(* CoDeSys 2.3.9.41 project: PLC.pro *)
(* Libraries: ModBus.lib 27.5.09 10:22:38, ComService.lib 21.5.09 15:28:28, SysLibCom.lib 20.2.06 14:31:08, STANDARD.LIB 4.10.05 11:14:46, IECSFC.LIB 13.4.06 15:51:28, SYSLIBTIME.LIB 20.2.06 14:31:16, SYSTASKINFO.LIB 20.2.06 14:31:38, ANALYZATION.LIB 5.10.99 09:05:06, Util.lib 18.5.10 15:14:28, SYSLIBCALLBACK.LIB 20.2.06 14:31:08 *)

(* PLC configuration (modules and I/O channels)
PDI1Q AT %IX0.0 [BitInput] Discrete input 1
PDI2Q AT %IX0.1 [BitInput] Discrete input 2
PDI3Q AT %IX0.2 [BitInput] Discrete input 3
PDI4Q AT %IX0.3 [BitInput] Discrete input 4
Discrete inputs [ID130] node 1, in %IB1 out %QB1 {Filtrationtime_GeneralINP = 10; Visibility = No; PinCount = 12}
  AT %IB1.0 [ByteInput] 8 discrete inputs
  AT %IB1.1 [ByteInput] 4 discrete inputs
Discrete outputs [ID131] node 2, in %IB2 out %QB2 {SafeValueByte = 0; SafeValueByteM = 0; Visibility = No; PinCount = 12}
  AT %QB2.0 [ByteOutput] 8 discrete outputs
  AT %QB2.1 [ByteOutput] 4 discrete outputs
Fast analog inputs [ID125] node 3, in %IB3 out %QB3 {Flt_Comm = 50Hz 2Por}
  AT %IR3.0 [FloatInputP] AI #1 {AIN_TYPE = 4-20 mA; Peak_Filtr = 200; Flt_Ch = Off; TauRC = 10; MinFV = 0; MaxFV = 20000.0}
  AT %IR3.1 [FloatInputP] AI #2 {AIN_TYPE = 4-20 mA; Peak_Filtr = 200; Flt_Ch = Off; TauRC = 10; MinFV = 0; MaxFV = 20000.0}
  AT %IR3.2 [FloatInputP] AI #3 {AIN_TYPE = 4-20 mA; Peak_Filtr = 200; Flt_Ch = Off; TauRC = 10; MinFV = 0; MaxFV = 20000.0}
  AT %IR3.3 [FloatInputP] AI #4 {AIN_TYPE = 4-20 mA; Peak_Filtr = 200; Flt_Ch = Off; TauRC = 10; MinFV = 0; MaxFV = 20000.0}
  AT %IR3.4 [FloatInputP] AI #5 {AIN_TYPE = 4-20 mA; Peak_Filtr = 200; Flt_Ch = Off; TauRC = 10; MinFV = 0; MaxFV = 20000.0}
  AT %IR3.5 [FloatInputP] AI #6 {AIN_TYPE = 4-20 mA; Peak_Filtr = 200; Flt_Ch = Off; TauRC = 10; MinFV = 0; MaxFV = 20000.0}
  AT %IR3.6 [FloatInputP] AI #7 {AIN_TYPE = 4-20 mA; Peak_Filtr = 200; Flt_Ch = Off; TauRC = 10; MinFV = 0; MaxFV = 20000.0}
  AT %IR3.7 [FloatInputP] AI #8 {AIN_TYPE = 4-20 mA; Peak_Filtr = 200; Flt_Ch = Off; TauRC = 10; MinFV = 0; MaxFV = 20000.0}
  AT %IW3.8 [WordInput] AI read time (10ms)
Analog outputs [ID126] node 4, in %IB4 out %QB4
  PAO01 AT %QR4.0 [FloatOutputP] AO #1 {AOUT_TYPE = 4-20 mA; SafeValueREAL = 0.0}
  AT %QR4.1 [FloatOutputP] AO #2 {AOUT_TYPE = 4-20 mA; SafeValueREAL = 0.0}
  AT %QR4.2 [FloatOutputP] AO #3 {AOUT_TYPE = 4-20 mA; SafeValueREAL = 0.0}
  AT %QR4.3 [FloatOutputP] AO #4 {AOUT_TYPE = 4-20 mA; SafeValueREAL = 0.0}
Special input [ID103] node 5, in %IB5 out %QB5 {Filtrationtime = 1000; PinCount = 1; WatchDogPeriod = 400; PollPeriod = 3000; Visibility = No}
  AT %IX5.0 [BitInput] Special input
Special output [ID104] node 6, in %IB6 out %QB6 {Visibility = No; PinCount = 1}
  AT %QX6.0 [BitOutput] Special output
Modbus [MODBUS_ID302] node 0, in %IB7.0 out %QB7.0
  TCP [TCP_ID221] node 0, in %IB7.0.0 out %QB7.0.0 {RemotePort = 502; Visibility = No}
  TCP [TCP_ID221] node 1, in %IB7.0.1 out %QB7.0.1 {RemotePort = 502; Visibility = No}
  TCP [TCP_ID221] node 2, in %IB7.0.2 out %QB7.0.2 {RemotePort = 504; Visibility = No}
  TCP [TCP_ID221] node 3, in %IB7.0.3 out %QB7.0.3 {RemotePort = 502; Visibility = No}
  TCP [TCP_ID221] node 4, in %IB7.0.4 out %QB7.0.4 {RemotePort = 502; Visibility = No}
  RS-232 [COM2_USART] node 5, in %IB7.0.5 out %QB7.0.5 {CommunicationSpeed = 11520; Parity = NO PARITY CHECK; BitLength = 8 bits; StopLength = One stop bit; InterfaceType = RS232; FrameOriented = RTU; Timeout = 0; Visibility = No}
  Debug RS-232 [DEBUG_USART] node 6, in %IB7.0.6 out %QB7.0.6 {CommunicationSpeed = 11520; Parity = NO PARITY CHECK; BitLength = 8 bits; StopLength = One stop bit; InterfaceType = RS232; FrameOriented = RTU; Timeout = 0; Visibility = No}
  TCP [TCP_ID221] node 7, in %IB7.0.7 out %QB7.0.7 {RemotePort = 502; Visibility = No}
  TCP [TCP_ID221] node 8, in %IB7.0.8 out %QB7.0.8 {RemotePort = 502; Visibility = No}
AT %QB7.1.0 [ByteOutput]
8 bits [8Bit] node 2, in %IB7.2 out %QB7.2
  AT %QB7.2.0 [ByteOutput]
8 bits [8Bit] node 3, in %IB7.3 out %QB7.3
  AT %QB7.3.0 [ByteOutput]
8 bits [8Bit] node 4, in %IB7.4 out %QB7.4
  AT %QB7.4.0 [ByteOutput]
  AT %QB7.5.0 [ByteOutput]
8 bits [8Bit] node 6, in %IB7.6 out %QB7.6
  AT %QB7.6.0 [ByteOutput]
  Bit 7 AT %QB7.7.0 [ByteOutput] Module.8Bit3Module.MODBUS_ID4008 bitsIB%QB%MB%M
8 bits [8Bit] node 8, in %IB7.8 out %QB7.8
  AT %QB7.8.0 [ByteOutput]
  AT %QB7.9.0 [ByteOutput]
  AT %QB7.10.0 [ByteOutput]
  AT %QB7.11.0 [ByteOutput]
  AT %QB7.12.0 [ByteOutput]
  AT %QB7.13.0 [ByteOutput]
  AT %QB7.14.0 [ByteOutput]
  AT %QB7.15.0 [ByteOutput]
  AT %QB7.16.0 [ByteOutput]
  AT %QB7.17.0 [ByteOutput]
  AT %QB7.18.0 [ByteOutput]
  AT %QB7.19.0 [ByteOutput]
  AT %QB7.20.0 [ByteOutput]
8 bits [8Bit] node 21, in %IB7.21 out %QB7.21
  AT %QB7.21.0 [ByteOutput]
8 bits [8Bit] node 22, in %IB7.22 out %QB7.22
  AT %QB7.22.0 [ByteOutput]
2 byte [Register] node 23, in %IB7.23 out %QB7.23
  L16001_CUR AT %QW7.23.0 [WordOutput]
2 byte [Register] node 24, in %IB7.24 out %QB7.24
  L16106_CUR AT %QW7.24.0 [WordOutput]
2 byte [Register] node 25, in %IB7.25 out %QB7.25
  X16106M1_CUR AT %QW7.25.0 [WordOutput]
2 byte [Register] node 26, in %IB7.26 out %QB7.26
  C16105_CUR AT %QW7.26.0 [WordOutput]
2 byte [Register] node 27, in %IB7.27 out %QB7.27
  M16105_PER AT %QW7.27.0 [WordOutput]
2 byte [Register] node 28, in %IB7.28 out %QB7.28
  C16103_CUR AT %QW7.28.0 [WordOutput]
2 byte [Register] node 29, in %IB7.29 out %QB7.29
  M16103_PER AT %QW7.29.0 [WordOutput]
2 byte [Register] node 30, in %IB7.30 out %QB7.30
  M16106_PV AT %QW7.30.0 [WordOutput]
2 byte [Register] node 31, in %IB7.31 out %QB7.31
  L16201_CUR AT %QW7.31.0 [WordOutput]
2 byte [Register] node 32, in %IB7.32 out %QB7.32
  X16105A_CUR AT %QW7.32.0 [WordOutput]
2 byte [Register] node 33, in %IB7.33 out %QB7.33
  X16105B_CUR AT %QW7.33.0 [WordOutput]
2 byte [Register] node 34, in %IB7.34 out %QB7.34
  C16104_CUR AT %QW7.34.0 [WordOutput]
2 byte [Register] node 35, in %IB7.35 out %QB7.35
  M16104_PER AT %QW7.35.0 [WordOutput]
2 byte [Register] node 36, in %IB7.36 out %QB7.36
  L16101_CUR AT %QW7.36.0 [WordOutput]
2 byte [Register] node 37, in %IB7.37 out %QB7.37
  TRM_1_1 AT %QW7.37.0 [WordOutput]
2 byte [Register] node 38, in %IB7.38 out %QB7.38
  TRM_1_2 AT %QW7.38.0 [WordOutput]
2 byte [Register] node 39, in %IB7.39 out %QB7.39
  TRM_1_3 AT %QW7.39.0 [WordOutput]
  TRM_1_4 AT %QW7.40.0 [WordOutput]
2 byte [Register] node 41, in %IB7.41 out %QB7.41
  TRM_1_5 AT %QW7.41.0 [WordOutput]
2 byte [Register] node 42, in %IB7.42 out %QB7.42
  TRM_1_6 AT %QW7.42.0 [WordOutput]
2 byte [Register] node 43, in %IB7.43 out %QB7.43
  TRM_1_7 AT %QW7.43.0 [WordOutput]
2 byte [Register] node 44, in %IB7.44 out %QB7.44
  TRM_1_8 AT %QW7.44.0 [WordOutput]
2 byte [Register] node 45, in %IB7.45 out %QB7.45
  TRM_2_1 AT %QW7.45.0 [WordOutput]
2 byte [Register] node 46, in %IB7.46 out %QB7.46
  TRM_2_2 AT %QW7.46.0 [WordOutput]
2 byte [Register] node 47, in %IB7.47 out %QB7.47
  TRM_2_3 AT %QW7.47.0 [WordOutput]
2 byte [Register] node 48, in %IB7.48 out %QB7.48
  TRM_2_4 AT %QW7.48.0 [WordOutput]
2 byte [Register] node 49, in %IB7.49 out %QB7.49
  TRM_2_5 AT %QW7.49.0 [WordOutput]
2 byte [Register] node 50, in %IB7.50 out %QB7.50
  TRM_2_6 AT %QW7.50.0 [WordOutput]
2 byte [Register] node 51, in %IB7.51 out %QB7.51
  TRM_2_7 AT %QW7.51.0 [WordOutput]
2 byte [Register] node 52, in %IB7.52 out %QB7.52
  TRM_2_8 AT %QW7.52.0 [WordOutput]
2 byte [Register] node 53, in %IB7.53 out %QB7.53
  K16001_P AT %QW7.53.0 [WordOutput]
2 byte [Register] node 54, in %IB7.54 out %QB7.54
  M_3_6 AT %QW7.54.0 [WordOutput]
2 byte [Register] node 55, in %IB7.55 out %QB7.55
  M_3_7 AT %QW7.55.0 [WordOutput]
2 byte [Register] node 56, in %IB7.56 out %QB7.56
  M16106_CUR AT %QW7.56.0 [WordOutput]
  M16106_SP AT %QW7.57.0 [WordOutput]
  AT %QW7.58.0 [WordOutput]
2 byte [Register] node 59, in %IB7.59 out %QB7.59
  AT %QW7.59.0 [WordOutput]
2 byte [Register] node 60, in %IB7.60 out %QB7.60
  AT %QW7.60.0 [WordOutput]
2 byte [Register] node 61, in %IB7.61 out %QB7.61
  AT %QW7.61.0 [WordOutput]
2 byte [Register] node 62, in %IB7.62 out %QB7.62
  AT %QW7.62.0 [WordOutput]
2 byte [Register] node 63, in %IB7.63 out %QB7.63
  AT %QW7.63.0 [WordOutput]
2 byte [Register] node 64, in %IB7.64 out %QB7.64
  AT %QW7.64.0 [WordOutput]
2 byte [Register] node 65, in %IB7.65 out %QB7.65
  AT %QW7.65.0 [WordOutput]
  FLOW_SP_1 AT %QW7.66.0 [WordOutput]
  FLOW_SP_2 AT %QW7.67.0 [WordOutput]
  FLOW_SP_3 AT %QW7.68.0 [WordOutput]
  FLOW_SP_4 AT %QW7.69.0 [WordOutput]
  SPEED_1 AT %QW7.70.0 [WordOutput]
  SPEED_2 AT %QW7.71.0 [WordOutput]
  SPEED_3 AT %QW7.72.0 [WordOutput]
  SPEED_4 AT %QW7.73.0 [WordOutput]
  PERSENT1 AT %QW7.74.0 [WordOutput]
  PERSENT2 AT %QW7.75.0 [WordOutput]
  PERSENT3 AT %QW7.76.0 [WordOutput]
  PERSENT4 AT %QW7.77.0 [WordOutput]
  FLOW_TOT AT %QW7.78.0 [WordOutput]
  PER_TOT AT %QW7.79.0 [WordOutput]
  FLOW_SP_TOT AT %QW7.80.0 [WordOutput]
8 bits [8Bit] node 81, in %IB7.81 out %QB7.81
  AT %QB7.81.0 [ByteOutput]
8 bits [8Bit] node 82, in %IB7.82 out %QB7.82
  AT %QB7.82.0 [ByteOutput]
  AT %QB7.83.0 [ByteOutput]
  AT %QB7.84.0 [ByteOutput]
FLOW_1 AT %QW7.85.0 [WordOutput]
FLOW_2 AT %QW7.86.0 [WordOutput]
FLOW_3 AT %QW7.87.0 [WordOutput]
FLOW_4 AT %QW7.88.0 [WordOutput]
counter_1 AT %QD7.89.0 [FloatOutput]
counter_2 AT %QD7.90.0 [FloatOutput]
counter_3 AT %QD7.91.0 [FloatOutput]
counter_4 AT %QD7.92.0 [FloatOutput]
count_hour1 AT %QW7.93.0 [WordOutput]
count_hour2 AT %QW7.94.0 [WordOutput]
count_hour3 AT %QW7.95.0 [WordOutput]
count_hour4 AT %QW7.96.0 [WordOutput]
count_TOTAL AT %QW7.97.0 [WordOutput]
ModBus (Master) [MODBUS_MASTER_ID450] node 8, in %IB8 out %QB8 {Visibility = No}
  AT %QD8.0 [DWordOutput] Last address
  AT %QW8.1 [WordOutput] Last error
  RS-485-1 [COM1_USART] node 0, in %IB8.0 out %QB8.0 {CommunicationSpeed = 9600; Parity = NO PARITY CHECK; BitLength = 8 bits; StopLength = One stop bit; InterfaceType = RS485; FrameOriented = RTU; Timeout = 0; Visibility = No}
AT %QB8.1.0 [ComChannel] Command (0xff - Start)
count1 AT %ID8.1.0.0 [DWordInput]
flow1 AT %ID8.1.1.0 [DWordInput]
flow_sp1 AT %QD8.1.2.0 [DWordOutput]
speed1 AT %ID8.1.3.0 [DWordInput]
start1 AT %QW8.1.4.0 [WordOutput]
STATUS1 AT %IW8.1.5.0 [WordInput]
AT %QB8.2.0 [ComChannel] Command (0xff - Start)
count2 AT %ID8.2.0.0 [DWordInput]
flow2 AT %ID8.2.1.0 [DWordInput]
flow_sp2 AT %QD8.2.2.0 [DWordOutput]
speed2 AT %ID8.2.3.0 [DWordInput]
start2 AT %QW8.2.4.0 [WordOutput]
STATUS2 AT %IW8.2.5.0 [WordInput]
AT %QB8.3.0 [ComChannel] Command (0xff - Start)
count3 AT %ID8.3.0.0 [DWordInput]
flow3 AT %ID8.3.1.0 [DWordInput]
flow_sp3 AT %QD8.3.2.0 [DWordOutput]
speed3 AT %ID8.3.3.0 [DWordInput]
start3 AT %QW8.3.4.0 [WordOutput]
STATUS3 AT %IW8.3.5.0 [WordInput]
AT %QB8.4.0 [ComChannel] Command (0xff - Start)
count4 AT %ID8.4.0.0 [DWordInput]
flow4 AT %ID8.4.1.0 [DWordInput]
flow_sp4 AT %QD8.4.2.0 [DWordOutput]
speed4 AT %ID8.4.3.0 [DWordInput]
start4 AT %QW8.4.4.0 [WordOutput]
STATUS4 AT %IW8.4.5.0 [WordInput]
Universal Modbus device [ID2000] node 5, in %IB8.5 out %QB8.5 {ModuleIP = 10:0:0:223; ServiceTimeout = 150; TCPport = 502; NetMode = Serial; ModuleSlaveAddress = 8; RequestType = Both; PeriodOfService = 10; Visibility = No; RepeatCounter = 0; ByteSequence = Trace_mode}
  AT %QB8.5.0 [ComChannel] Command (0xff - Start)
MDI_1_0 AT %IW8.5.0.0 [WordInput]
MDI_1_1 AT %IW8.5.1.0 [WordInput]
Universal Modbus device [ID2000] node 6, in %IB8.6 out %QB8.6 {ModuleIP = 10:0:0:223; ServiceTimeout = 150; TCPport = 502; NetMode = Serial; ModuleSlaveAddress = 16; RequestType = Both; PeriodOfService = 10; Visibility = No; RepeatCounter = 0; ByteSequence = Trace_mode}
  AT %QB8.6.0 [ComChannel] Command (0xff - Start)
MDI_2_0 AT %IW8.6.0.0 [WordInput]
MDI_2_1 AT %IW8.6.1.0 [WordInput]
Universal Modbus device [ID2000] node 7, in %IB8.7 out %QB8.7 {ModuleIP = 10:0:0:223; ServiceTimeout = 150; TCPport = 502; NetMode = Serial; ModuleSlaveAddress = 24; RequestType = Both; PeriodOfService = 10; Visibility = No; RepeatCounter = 0; ByteSequence = Trace_mode}
  AT %QB8.7.0 [ComChannel] Command (0xff - Start)
MDI_3_0 AT %IW8.7.0.0 [WordInput]
MDI_3_1 AT %IW8.7.1.0 [WordInput]
Universal Modbus device [ID2000] node 8, in %IB8.8 out %QB8.8 {ModuleIP = 10:0:0:223; ServiceTimeout = 150; TCPport = 502; NetMode = Serial; ModuleSlaveAddress = 32; RequestType = Both; PeriodOfService = 10; Visibility = No; RepeatCounter = 0; ByteSequence = Trace_mode}
  AT %QB8.8.0 [ComChannel] Command (0xff - Start)
MDI_4_0 AT %IW8.8.0.0 [WordInput]
MDI_4_1 AT %IW8.8.1.0 [WordInput]
Universal Modbus device [ID2000] node 9, in %IB8.9 out %QB8.9 {ModuleIP = 10:0:0:223; ServiceTimeout = 150; TCPport = 502; NetMode = Serial; ModuleSlaveAddress = 40; RequestType = Both; PeriodOfService = 10; Visibility = No; RepeatCounter = 0; ByteSequence = Trace_mode}
  AT %QB8.9.0 [ComChannel] Command (0xff - Start)
MDO1_0 AT %QW8.9.0.0 [WordOutput]
MDO1_1 AT %QW8.9.1.0 [WordOutput]
MDO1_2 AT %QW8.9.2.0 [WordOutput]
MDO1_3 AT %QW8.9.3.0 [WordOutput]
MDO1_4 AT %QW8.9.4.0 [WordOutput]
MDO1_5 AT %QW8.9.5.0 [WordOutput]
MDO1_6 AT %QW8.9.6.0 [WordOutput]
MDO1_7 AT %QW8.9.7.0 [WordOutput]
MDO1_8 AT %QW8.9.8.0 [WordOutput]
MDO1_9 AT %QW8.9.9.0 [WordOutput]
MDO1_10 AT %QW8.9.10.0 [WordOutput]
MDO1_11 AT %QW8.9.11.0 [WordOutput]
MDO1_12 AT %QW8.9.12.0 [WordOutput]
MDO1_13 AT %QW8.9.13.0 [WordOutput]
MDO1_14 AT %QW8.9.14.0 [WordOutput]
MDO1_15 AT %QW8.9.15.0 [WordOutput]
Universal Modbus device [ID2000] node 10, in %IB8.10 out %QB8.10 {ModuleIP = 10:0:0:223; ServiceTimeout = 150; TCPport = 502; NetMode = Serial; ModuleSlaveAddress = 48; RequestType = Both; PeriodOfService = 10; Visibility = No; RepeatCounter = 0; ByteSequence = Trace_mode}
  AT %QB8.10.0 [ComChannel] Command (0xff - Start)
MDO2_0 AT %QW8.10.0.0 [WordOutput]
MDO2_1 AT %QW8.10.1.0 [WordOutput]
MDO2_2 AT %QW8.10.2.0 [WordOutput]
MDO2_3 AT %QW8.10.3.0 [WordOutput]
MDO2_4 AT %QW8.10.4.0 [WordOutput]
MDO2_5 AT %QW8.10.5.0 [WordOutput]
MDO2_6 AT %QW8.10.6.0 [WordOutput]
MDO2_7 AT %QW8.10.7.0 [WordOutput]
MDO2_8 AT %QW8.10.8.0 [WordOutput]
MDO2_9 AT %QW8.10.9.0 [WordOutput]
MDO2_10 AT %QW8.10.10.0 [WordOutput]
MDO2_11 AT %QW8.10.11.0 [WordOutput]
MDO2_12 AT %QW8.10.12.0 [WordOutput]
MDO2_13 AT %QW8.10.13.0 [WordOutput]
MDO2_14 AT %QW8.10.14.0 [WordOutput]
MDO2_15 AT %QW8.10.15.0 [WordOutput]
Universal Modbus device [ID2000] node 11, in %IB8.11 out %QB8.11 {ModuleIP = 10:0:0:223; ServiceTimeout = 150; TCPport = 502; NetMode = Serial; ModuleSlaveAddress = 56; RequestType = Both; PeriodOfService = 10; Visibility = No; RepeatCounter = 0; ByteSequence = Trace_mode}
  AT %QB8.11.0 [ComChannel] Command (0xff - Start)
M1_1 AT %IW8.11.0.0 [WordInput]
M1_2 AT %IW8.11.1.0 [WordInput]
M1_3 AT %IW8.11.2.0 [WordInput]
M1_4 AT %IW8.11.3.0 [WordInput]
M1_5 AT %IW8.11.4.0 [WordInput]
M1_6 AT %IW8.11.5.0 [WordInput]
M1_7 AT %IW8.11.6.0 [WordInput]
M1_8 AT %IW8.11.7.0 [WordInput]
Universal Modbus device [ID2000] node 12, in %IB8.12 out %QB8.12 {ModuleIP = 10:0:0:223; ServiceTimeout = 150; TCPport = 502; NetMode = Serial; ModuleSlaveAddress = 64; RequestType = Both; PeriodOfService = 10; Visibility = No; RepeatCounter = 0; ByteSequence = Trace_mode}
  AT %QB8.12.0 [ComChannel] Command (0xff - Start)
M2_1 AT %IW8.12.0.0 [WordInput]
M2_2 AT %IW8.12.1.0 [WordInput]
M2_3 AT %IW8.12.2.0 [WordInput]
M2_4 AT %IW8.12.3.0 [WordInput]
M2_5 AT %IW8.12.4.0 [WordInput]
M2_6 AT %IW8.12.5.0 [WordInput]
M2_7 AT %IW8.12.6.0 [WordInput]
M2_8 AT %IW8.12.7.0 [WordInput]
Universal Modbus device [ID2000] node 13, in %IB8.13 out %QB8.13 {ModuleIP = 10:0:0:223; ServiceTimeout = 150; TCPport = 502; NetMode = Serial; ModuleSlaveAddress = 72; RequestType = Both; PeriodOfService = 10; Visibility = No; RepeatCounter = 0; ByteSequence = Trace_mode}
  AT %QB8.13.0 [ComChannel] Command (0xff - Start)
M3_1 AT %IW8.13.0.0 [WordInput]
M3_2 AT %IW8.13.1.0 [WordInput]
M3_3 AT %IW8.13.2.0 [WordInput]
M3_4 AT %IW8.13.3.0 [WordInput]
M3_5 AT %IW8.13.4.0 [WordInput]
M3_6 AT %IW8.13.5.0 [WordInput]
M3_7 AT %IW8.13.6.0 [WordInput]
M3_8 AT %IW8.13.7.0 [WordInput]
Universal Modbus device [ID2000] node 14, in %IB8.14 out %QB8.14 {ModuleIP = 10:0:0:223; ServiceTimeout = 150; TCPport = 502; NetMode = Serial; ModuleSlaveAddress = 80; RequestType = Both; PeriodOfService = 10; Visibility = No; RepeatCounter = 0; ByteSequence = Trace_mode}
  AT %QB8.14.0 [ComChannel] Command (0xff - Start)
TRM_1_1_RS AT %ID8.14.0.0 [FloatInput]
TRM_1_2_RS AT %ID8.14.1.0 [FloatInput]
TRM_1_3_RS AT %ID8.14.2.0 [FloatInput]
TRM_1_4_RS AT %ID8.14.3.0 [FloatInput]
TRM_1_5_RS AT %ID8.14.4.0 [FloatInput]
TRM_1_6_RS AT %ID8.14.5.0 [FloatInput]
TRM_1_7_RS AT %ID8.14.6.0 [FloatInput]
TRM_1_8_RS AT %ID8.14.7.0 [FloatInput]
Universal Modbus device [ID2000] node 15, in %IB8.15 out %QB8.15 {ModuleIP = 10:0:0:223; ServiceTimeout = 150; TCPport = 502; NetMode = Serial; ModuleSlaveAddress = 88; RequestType = Both; PeriodOfService = 10; Visibility = No; RepeatCounter = 0; ByteSequence = Trace_mode}
  AT %QB8.15.0 [ComChannel] Command (0xff - Start)
TRM_2_1_RS AT %ID8.15.0.0 [FloatInput]
TRM_2_2_RS AT %ID8.15.1.0 [FloatInput]
TRM_2_3_RS AT %ID8.15.2.0 [FloatInput]
TRM_2_4_RS AT %ID8.15.3.0 [FloatInput]
TRM_2_5_RS AT %ID8.15.4.0 [FloatInput]
TRM_2_6_RS AT %ID8.15.5.0 [FloatInput]
TRM_2_7_RS AT %ID8.15.6.0 [FloatInput]
TRM_2_8_RS AT %ID8.15.7.0 [FloatInput]
Button [ID003] node 9, in %IB9 out %QB9
  AT %IX9.0 [BitInput] Button Start/Stop
*)

(* Global variable list: Global_Variables *)
VAR_GLOBAL
	L16003_SRT_G : BOOL;
	X16011_SRT_G : BOOL;
	L16106_SRT_G : BOOL;
	L16004_SRT_G : BOOL;
	X16011_A_SRT_G : BOOL;
	X16106M1_SRT_G : BOOL;
	X16106M1_STP_G : BOOL;
	X16106MA_SRT_G : BOOL;
	X16106MB_SRT_G : BOOL;
	X16106M2_SRT_G : BOOL;
	O161061_SRT_G : BOOL;
	O161062_SRT_G : BOOL;
	O161063_SRT_G : BOOL;
	O161064_SRT_G : BOOL;
	C16101_SRT_G : BOOL;
	C16105_SRT_G : BOOL;
	(*********************************)
	M16105_OPN_G : BOOL;
	M16105_CLS_G : BOOL;
	C16103_SRT_G : BOOL;
	M16103_OPN_G : BOOL;
	M16103_CLS_G : BOOL;
	C16106_SRT_G : BOOL;
	L16107_SRT_G : BOOL;
	M16106_SRT_G : BOOL;
	O16106_SRT_G : BOOL;
	B16401_SRT_G : BOOL;
	B16402_SRT_G : BOOL;
	X16106M1_G : BOOL;
	B16404_SRT_G : BOOL;
	L16005_SRT_G : BOOL;

	L16201_SRT_G : BOOL;
	C16201_SRT_G : BOOL;
	(*****************************)
	C16104_SRT_G : BOOL;
	L16101_SRT_G : BOOL;
	X16106M1_FAZA_G : BOOL;

END_VAR
VAR_GLOBAL RETAIN PERSISTENT

	eski_counter_1: REAL;
	eski_counter_2: REAL;
	eski_counter_3: REAL;
	eski_counter_4: REAL;


END_VAR

(* POU PLC_PRG, ST *)
PROGRAM PLC_PRG
VAR
END_VAR
TRANSLATE();
ALARM_RPM();
(*BLOCK();*)
vaqt();
END_PROGRAM

(* POU TRANSLATE, ST *)
PROGRAM TRANSLATE
VAR
	B164: BOOL;
	MA : ARRAY [1..30] OF MY_LINTRAFO;
	RTRIG: R_TRIG;
	FTRIG: F_TRIG;

	FLOW_ZAD: BOOL;
	FLOW_ZAD_1: BOOL;
	FLOW_ZAD_2: BOOL;
	FLOW_ZAD_3: BOOL;
	FLOW_ZAD_4: BOOL;
	f: BOOL;

	PAO01_TMP: WORD;
END_VAR
OUTPUTS();
MDI1_0();
MDI1_1();
MDI2_0();
MDI2_1();
MDI3_0();
MDI3_1();
MDI4_0();
MDI4_1();


DOZ();
BLOCK();
 M16106_SP := LIMIT(10, M16106_SP, 50);
MA[30](IN := M16106_SP,  IN_MIN := 10, IN_MAX :=50 , OUT_MIN := 4.0,  OUT_MAX := 20.0, OUT => PAO01_TMP);
PAO01 := PAO01_TMP / 100.0;
MA[1](IN := M1_1, IN_MIN := 400.0, IN_MAX := 2000.0, OUT_MIN := 0.0,  OUT_MAX := 200.0, OUT => L16001_CUR);
MA[2](IN := M1_2,  OUT_MIN := 0.0,  OUT_MAX := 200.0, OUT => L16106_CUR);
MA[3](IN := M1_7, IN_MIN := 400.0, IN_MAX := 2000.0, OUT_MIN := 0.0,  OUT_MAX := 290.0, OUT => X16106M1_CUR);
MA[4](IN := M1_3, OUT_MIN := 0.0,  OUT_MAX := 200.0, OUT => C16105_CUR);
MA[5](IN := M1_4, IN_MIN := 800, IN_MAX := 2000,  OUT_MIN := 0.0,  OUT_MAX := 100.0, OUT => M16105_PER);
MA[6](IN := M2_7, OUT_MIN :=0.0,  OUT_MAX := 100.0, OUT => C16103_CUR);
MA[7](IN := M2_8, OUT_MIN := 0.0,  OUT_MAX := 100.0, OUT => M16103_PER);
MA[8](IN := M1_6,  IN_MIN := 400.0, IN_MAX := 2000.0, OUT_MIN := 0.0,  OUT_MAX := 50.0, OUT => M16106_CUR);
MA[9](IN := M2_1, OUT_MIN := 0.0,  OUT_MAX := 200.0, OUT => L16201_CUR);
MA[10](IN := M2_4, OUT_MIN := 0.0,  OUT_MAX := 200.0, OUT =>C16104_CUR);
MA[11](IN := M2_5,  IN_MIN := 0.0, IN_MAX := 100.0, OUT_MIN := 0.0,  OUT_MAX := 100.0, OUT => M16104_PER);
MA[12](IN := M2_6, OUT_MIN := 0.0,  OUT_MAX := 200.0, OUT => L16101_CUR);
MA[17](IN := M1_8, IN_MIN := 400.0, IN_MAX := 2000.0, OUT_MIN := 0.0,  OUT_MAX := 496.0, OUT => M16106_PV);
TRM_1_1 := REAL_TO_WORD( TRM_1_1_RS * 100);
TRM_1_2 := REAL_TO_WORD(TRM_1_2_RS * 100);
TRM_1_3 := REAL_TO_WORD(TRM_1_3_RS * 100);
TRM_1_4 := REAL_TO_WORD(TRM_1_4_RS * 100);
TRM_1_5 := REAL_TO_WORD(TRM_1_5_RS * 100);
TRM_1_6 := REAL_TO_WORD(TRM_1_6_RS * 100);
TRM_1_7 := REAL_TO_WORD(TRM_1_7_RS * 100);
TRM_1_8 := REAL_TO_WORD(TRM_1_8_RS * 100);

TRM_2_1 := REAL_TO_WORD(TRM_2_1_RS * 100);
TRM_2_2 := REAL_TO_WORD(TRM_2_2_RS * 100);
TRM_2_3 := REAL_TO_WORD(TRM_2_3_RS * 100);
TRM_2_4 := REAL_TO_WORD(TRM_2_4_RS * 100);
TRM_2_5 := REAL_TO_WORD(TRM_2_5_RS * 100);
TRM_2_6 := REAL_TO_WORD(TRM_2_6_RS * 100);
TRM_2_7 := REAL_TO_WORD(TRM_2_7_RS * 100);
TRM_2_8 := REAL_TO_WORD(TRM_2_8_RS * 100);


MA[13](IN := M3_5, OUT_MIN := 0,  OUT_MAX := 16, OUT => K16001_P);
MA[14](IN := M3_6, OUT_MIN := -10,  OUT_MAX := 10.0, OUT => M_3_6);
MA[15](IN := M3_7, OUT_MIN := -10,  OUT_MAX := 10.0, OUT => M_3_7);
(*
MA[16](IN := M3_8, OUT_MIN := 0.0,  OUT_MAX := 1000.0, OUT => M16106_PV);*)
END_PROGRAM
ACTION DOZ:
W16001_WRK  := WORD_TO_BOOL(STATUS1 MOD 2);
W16002_WRK  := WORD_TO_BOOL(STATUS2 MOD 2);
W16003_WRK  := WORD_TO_BOOL(STATUS3 MOD 2);
W16004_WRK  := WORD_TO_BOOL(STATUS4 MOD 2);

FLOW_TOT := DWORD_TO_WORD((flow1 + flow2 + flow3 + flow4)/100);
PER_TOT := PERSENT1 + PERSENT2 + PERSENT3 + PERSENT4;
SPEED_1 := DWORD_TO_WORD(speed1);
SPEED_2 := DWORD_TO_WORD(speed2);
SPEED_3 := DWORD_TO_WORD(speed3);
SPEED_4 := DWORD_TO_WORD(speed4);
FLOW_SP_1 := DWORD_TO_WORD(flow_sp1/100);
FLOW_SP_2 := DWORD_TO_WORD(flow_sp2/100);
FLOW_SP_3 := DWORD_TO_WORD(flow_sp3/100);
FLOW_SP_4 := DWORD_TO_WORD(flow_sp4/100);

FLOW_1 := DWORD_TO_WORD(flow1/100);
FLOW_2 := DWORD_TO_WORD(flow2/100);
FLOW_3 := DWORD_TO_WORD(flow3/100);
FLOW_4 := DWORD_TO_WORD(flow4/100);

counter_1 := DWORD_TO_REAL(count1)/1000 ;
counter_2 :=  DWORD_TO_REAL(count2)/1000 ;
counter_3 :=  DWORD_TO_REAL(count3)/1000;
counter_4 :=  DWORD_TO_REAL(count4)/1000;


(*FLOW_SP_TOT := DWORD_TO_WORD( flow_sp1 + flow_sp2 + flow_sp3 + flow_sp4);*)

IF (DOZ_CONF = TRUE AND PER_TOT = 10000)  THEN
	flow_sp1 := FLOW_SP_TOT * PERSENT1/ 1000;
	flow_sp2 := FLOW_SP_TOT * PERSENT2/1000;
	flow_sp3 := FLOW_SP_TOT * PERSENT3/1000;
	flow_sp4 := FLOW_SP_TOT * PERSENT4/1000;
	DOZ_CONF := FALSE;
END_IF;
RTRIG(CLK := DOZ_STR);
IF (L16003_BLK = FALSE AND L16003_WRK = FALSE) THEN
	DOZ_STR := FALSE;
END_IF;
(*IF (RTRIG.Q = TRUE (*AND L16003_BLK*)) THEN*)
(*
IF (DOZ_STR = TRUE (*AND L16003_BLK*)) THEN
	start1 := BOOL_TO_WORD(PERSENT1 > 0 AND L16003_WRK) ;
	start2 := BOOL_TO_WORD(PERSENT2 > 0 AND L16003_WRK)  ;
	start3 := BOOL_TO_WORD(PERSENT3 > 0 AND L16003_WRK)  ;
	start4 := BOOL_TO_WORD(PERSENT4 > 0 AND L16003_WRK) ;
END_IF;*)
IF (DOZ_STR = TRUE (*AND L16003_BLK*)) THEN
	IF STATUS1 = 4 THEN
		start1 := BOOL_TO_WORD(PERSENT1 > 0 ) ;
	ELSE
		START1 := 5;
	END_IF;

	IF STATUS2 = 4 THEN
		start2 := BOOL_TO_WORD(PERSENT2 > 0 ) ;
	ELSE
		START2 := 5;
	END_IF;

	IF STATUS3 = 4 THEN
		start3 := BOOL_TO_WORD(PERSENT3 > 0 ) ;
	ELSE
		START3 := 5;
	END_IF;

	IF STATUS4 = 4 THEN
		start4 := BOOL_TO_WORD(PERSENT4 > 0 ) ;
	ELSE
		START4 := 5;
	END_IF;
END_IF;
FTRIG( CLK := DOZ_STR);
(*IF (FTRIG.Q = TRUE )THEN*)
IF (DOZ_STR = FALSE)THEN
	start1 := 0;
	start2 := 0;
	start3 := 0;
	start4 := 0;
END_IF;
END_ACTION
ACTION MDI1_0:
W15001_1 := MDI_1_0.0;
W15001_2 := MDI_1_0.1;
W15001_3 := MDI_1_0.2;
W15001_4 := MDI_1_0.3;
W15001_5 := MDI_1_0.4;
W15001_6 := MDI_1_0.5;
W15001_7 := MDI_1_0.6;
W15001_8 := MDI_1_0.7;
W15001_9 := MDI_1_0.8;
W15001_10 := MDI_1_0.9;
W15001_11 := MDI_1_0.10;
L15003_WRK := MDI_1_0.12;
L15005_WRK := MDI_1_0.13;
L16001_WRK := MDI_1_0.14;
L16002_WRK := MDI_1_0.15;
END_ACTION
ACTION MDI1_1:
L16002_A_POS_1 := MDI_1_1.0;
L16002_A_POS_2 := MDI_1_1.1;
L16002_B_POS_1 := MDI_1_1.2;
L16002_B_POS_2 := MDI_1_1.3;
L16002_C_POS_1 := MDI_1_1.4;
L16002_C_POS_2 := MDI_1_1.5;
L16003_REM := MDI_1_1.6;
L16003_WRK := MDI_1_1.7;
X16011_REM := MDI_1_1.8;
X16011_WRK := MDI_1_1.9;
L16106_REM := MDI_1_1.10;
L16106_WRK := MDI_1_1.11;
L16004_REM := MDI_1_1.12;
L16004_WRK := MDI_1_1.13;
X16011_A_REM:= MDI_1_1.14;
X16011_A_WRK := MDI_1_1.15;
END_ACTION
ACTION MDI2_0:
X16106M1_REM := MDI_2_0.0;
X16106M1_QF_POL := NOT  MDI_2_0.1;
X16106M1_QF_RDY := MDI_2_0.2;
X16106MA_REM := MDI_2_0.3;
X16106MA_WRK := MDI_2_0.4;
X16106MB_REM := MDI_2_0.5;
X16106MB_WRK := MDI_2_0.6;
X16106M1_SH1_2_RDY := MDI_2_0.7;
X16106M1_EN := MDI_2_0.8;
O161061_REM := MDI_2_0.9;
O161061_PUMP1 := MDI_2_0.10;
O161061_PUMP2 := MDI_2_0.11;
C16103T := MDI_2_0.12;
O161061_RDY := MDI_2_0.13;
O161062_REM := MDI_2_0.14;
O161062_PUMP1 := MDI_2_0.15;
END_ACTION
ACTION MDI2_1:
O161062_PUMP2 := MDI_2_1.0;
C16104T := MDI_2_1.1;
O161062_RDY := MDI_2_1.2;
O161064_REM := MDI_2_1.3;
O161064_PUMP1 := MDI_2_1.4;
O161064_PUMP2 := MDI_2_1.5;
O161064_PUMP3 := MDI_2_1.6;
O161064_RDY := MDI_2_1.7;
O161063_REM := MDI_2_1.8;
O161063_PUMP1 := MDI_2_1.9;
O161063_PUMP2 := MDI_2_1.10;
O161063_PUMP3 := MDI_2_1.11;
O161063_RDY := MDI_2_1.12;
C16101_REM :=  MDI_2_1.13;
C16101_WRK := MDI_2_1.14;
C16105_REM := MDI_2_1.15;
END_ACTION
ACTION MDI3_0:
C16105_WRK := MDI_3_0.0;
M16105_REM := MDI_3_0.1;
X16108_WRK := MDI_3_0.2;
C16103_REM := MDI_3_0.3;
C16103_WRK :=  NOT MDI_3_0.4;
M16103_REM := MDI_3_0.5;
X16107_WRK := MDI_3_0.6;
C16106_REM := MDI_3_0.7;
C16106_WRK := MDI_3_0.8;
L16107_REM := MDI_3_0.9;
L16107_WRK := MDI_3_0.10;
M16106_REM := MDI_3_0.11;
M16106_WRK := MDI_3_0.12;
O16106_REM := MDI_3_0.13;
O16106_PUMP1 := MDI_3_0.14;
O16106_PUMP2 := MDI_3_0.15;
END_ACTION
ACTION MDI3_1:
O16106_RDY :=  MDI_3_1.0;
B16401_REM := MDI_3_1.1;
B16401_WRK := MDI_3_1.2;
B16402_REM := MDI_3_1.3;
B16402_WRK := MDI_3_1.4;
B16403_OPN := MDI_3_1.5;
B16403_CLS := MDI_3_1.6;
B16404_REM := MDI_3_1.7;
B16404_WRK := MDI_3_1.8;
B16405_OPN := MDI_3_1.9;
B16405_CLS := MDI_3_1.10;
L16201_REM := MDI_3_1.11;
L16201_WRK := MDI_3_1.12;
C16201_REM := MDI_3_1.13;
C16201_WRK := MDI_3_1.14;
C16201_A_REM := MDI_3_1.15;
END_ACTION
ACTION MDI4_0:
C16201_A_POS_1 := MDI_4_0.0;
C16201_A_POS_2 := MDI_4_0.1;
C16201_B_REM := MDI_4_0.2;
C16201_B_POS_1 := MDI_4_0.3;
C16201_B_POS_2 := MDI_4_0.4;
X16105_A_WRK := MDI_4_0.5;
X16105_B_WRK  := MDI_4_0.6;
C16104_REM := MDI_4_0.7;
C16104_WRK := NOT  MDI_4_0.8;
M16104_REM := MDI_4_0.9;
L16101_REM := MDI_4_0.10;
L16101_WRK := MDI_4_0.11;
L16101_REM := MDI_4_0.10;
L16101_WRK := MDI_4_0.11;
L16102_REM := MDI_4_0.12;
L16102_WRK := MDI_4_0.13;
TEMP_REDUC := MDI_4_0.14;
(*
RESET_BOX := MDI_4_0.15;*)
END_ACTION
ACTION MDI4_1:
C16103_RDY := MDI_4_1.0;
C16104_RDY := MDI_4_1.1;
L16005_REM := MDI_4_1.2;
L16005_WRK := MDI_4_1.3;
X16106M1_FZ_EN := MDI_4_1.4;
X16106M1_RP3 :=  MDI_4_1.5;
X16106M1_SHK1 := NOT  MDI_4_1.6;
X16106M1_ER :=NOT  MDI_4_1.7;
END_ACTION
ACTION OUTPUTS:
(********************************************************)
MDO1_0 := BOOL_TO_WORD( L16003_SRT_G) * 1000;  (*&*)
MDO1_1 := BOOL_TO_WORD( X16011_SRT_G ) * 1000;  (*&*)
MDO1_2 := BOOL_TO_WORD(L16106_SRT_G) * 1000; (*&*)
MDO1_3 := BOOL_TO_WORD( L16004_SRT_G) * 1000;  (*&*)
MDO1_4 := BOOL_TO_WORD( X16011_A_SRT_G) * 1000; (*&*)
MDO1_5 := BOOL_TO_WORD( X16106M1_SRT_G) * 1000;  (*&*)
(* MDO1_6 RESERV *)
MDO1_7 := BOOL_TO_WORD(X16106MA_SRT_G ) * 1000; (*&*)
MDO1_8 := BOOL_TO_WORD( X16106MB_SRT_G) * 1000; (*&&*)
MDO1_9 := BOOL_TO_WORD( X16106M2_SRT_G) * 1000; (*&&*)
MDO1_10 := BOOL_TO_WORD(O161061_SRT_G ) * 1000;  (*&*)
MDO1_11 := BOOL_TO_WORD(O161062_SRT_G ) * 1000; (*&*)
MDO1_12 := BOOL_TO_WORD(O161064_SRT_G) * 1000;  (*&*)
MDO1_13 := BOOL_TO_WORD(O161063_SRT_G) * 1000; (*&&*)
MDO1_14 := BOOL_TO_WORD(C16101_SRT_G ) * 1000; (*&*)
MDO1_15 := BOOL_TO_WORD(C16105_SRT ) * 1000; (*&*)
(***********************************************************)
MDO2_0 := BOOL_TO_WORD(M16105_OPN) * 1000;
MDO2_1 := BOOL_TO_WORD(M16105_CLS) * 1000;
MDO2_2 := BOOL_TO_WORD(C16103_SRT_G) * 1000; (*&*)
MDO2_3 := BOOL_TO_WORD(M16103_OPN) * 1000;
MDO2_4 := BOOL_TO_WORD(M16103_CLS) * 1000;
MDO2_5 := BOOL_TO_WORD(C16106_SRT_G) * 1000; (*&*)
MDO2_6 := BOOL_TO_WORD(L16107_SRT_G) * 1000;  (*&*)
MDO2_7 := BOOL_TO_WORD(M16106_SRT_G) * 1000; (*&*)
MDO2_8 := BOOL_TO_WORD(O16106_SRT_G) * 1000; (*&*)
MDO2_9 := BOOL_TO_WORD(B16401_SRT_G) * 1000; (*&*)
MDO2_10 := BOOL_TO_WORD(B16402_SRT_G) * 1000; (*&*)
MDO2_11 := BOOL_TO_WORD(X16106M1_FAZA_G) * 1000; (*###################*)
MDO2_12 := BOOL_TO_WORD(B16404_SRT_G) * 1000;
MDO2_13 := BOOL_TO_WORD( L16005_SRT_G) * 1000;  (*&*)
MDO2_14 := BOOL_TO_WORD(L16201_SRT_G ) * 1000;  (*&*)
MDO2_15 := BOOL_TO_WORD( C16201_SRT_G) * 1000; (*&*)
(*******************************************************

MDO1_0 := BOOL_TO_WORD( L16003_SRT) * 1000;
MDO1_1 := BOOL_TO_WORD( X16011_SRT ) * 1000;
MDO1_2 := BOOL_TO_WORD(L16106_SRT) * 1000;
MDO1_3 := BOOL_TO_WORD( L16004_SRT) * 1000;
MDO1_4 := BOOL_TO_WORD( X16011_A_SRT) * 1000;
MDO1_5 := BOOL_TO_WORD( X16106M1_SRT) * 1000;
MDO1_6 := BOOL_TO_WORD(X16106M1_STP ) * 1000;
MDO1_7 := BOOL_TO_WORD(X16106MA_SRT ) * 1000;
MDO1_8 := BOOL_TO_WORD( X16106MB_SRT) * 1000;
MDO1_9 := BOOL_TO_WORD( X16106M2_SRT) * 1000;
MDO1_10 := BOOL_TO_WORD(O161061_SRT) * 1000;
MDO1_11 := BOOL_TO_WORD(O161062_SRT ) * 1000;
MDO1_12 := BOOL_TO_WORD(O161064_SRT) * 1000;
MDO1_13 := BOOL_TO_WORD(O161063_SRT ) * 1000;
MDO1_14 := BOOL_TO_WORD(C16101_SRT ) * 1000;
MDO1_15 := BOOL_TO_WORD(C16105_SRT ) * 1000;
(*************************************************************)
MDO2_0 := BOOL_TO_WORD(M16105_OPN) * 1000;
MDO2_1 := BOOL_TO_WORD(M16105_CLS) * 1000;
MDO2_2 := BOOL_TO_WORD(C16103_SRT) * 1000;
MDO2_3 := BOOL_TO_WORD(M16103_OPN) * 1000;
MDO2_4 := BOOL_TO_WORD(M16103_CLS) * 1000;
MDO2_5 := BOOL_TO_WORD(C16106_SRT) * 1000;
MDO2_6 := BOOL_TO_WORD(L16107_SRT) * 1000;
MDO2_7 := BOOL_TO_WORD(M16106_SRT) * 1000;
MDO2_8 := BOOL_TO_WORD(O16106_SRT) * 1000;
MDO2_9 := BOOL_TO_WORD(B16401_SRT) * 1000;
MDO2_10 := BOOL_TO_WORD(B16402_SRT) * 1000;
MDO2_11 := BOOL_TO_WORD(X16106M1_FAZA ) * 1000;
MDO2_12 := BOOL_TO_WORD(B16404_SRT) * 1000;
MDO2_13 := BOOL_TO_WORD( L16005_SRT) * 1000;
MDO2_14 := BOOL_TO_WORD(L16201_SRT ) * 1000;
MDO2_15 := BOOL_TO_WORD( C16201_SRT) * 1000;

*****************************************************)
PDO1 := C16201_A_SRT;
PDO2 := C16201_B_SRT;
PDO3 := C16104_SRT_G; (*&*)
PDO4 := M16104_OPN;
PDO5 := M16104_CLS;
PDO6 := L16101_SRT_G;
PDO7 := L16102_SRT;
 W_HORN := PDO9;
PDO10 := C16103_STP; 		(*&*)
PDO11 := C16104_STP;		 (*&*)
PDO12 :=X16106M1_STP_G;
END_ACTION

(* POU MY_LINTRAFO, CFC *)
FUNCTION_BLOCK MY_LINTRAFO
VAR_INPUT
	IN : WORD;
	IN_MIN : REAL := 400.0;
	IN_MAX : REAL := 2000.0;
	OUT_MIN : REAL := 4.0;
	OUT_MAX : REAL := 20.0;
END_VAR
VAR_OUTPUT
	OUT : INT;
END_VAR
VAR
	LIN: LIN_TRAFO;
END_VAR
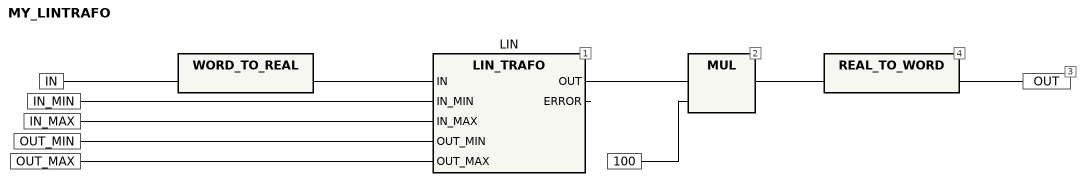
_CFC_ (* Continuous Function Chart, elements in execution order *)
#0 WORD_TO_REAL(IN)
#1 LIN:LIN_TRAFO(IN: #0, IN_MIN: IN_MIN, IN_MAX: IN_MAX, OUT_MIN: OUT_MIN, OUT_MAX: OUT_MAX)
#2 MUL(#1.OUT, 100)
#3 OUT <= #4
#4 REAL_TO_WORD(#2)
_END_CFC_
END_FUNCTION_BLOCK

(* POU BLOCK, LD *)
PROGRAM BLOCK
VAR
	R3 : BOOL;
	TP_WARING: TP;
	R_TR :  ARRAY [0..32] OF  R_TRIGs;
	F_TR :  ARRAY [0..32] OF  F_TRIGs;
	tonMEO : ARRAY[1..6] OF TON;
	VAQT : TIME := T#20s;
	vaqt2 : TIME := T#3s;
	vaqt3 : TIME := T#10s;
	vaqtMEO: TIME := T#2s;
	vaqt4 : TIME := T#30s;
	vaqtF : TIME := T#500ms;
	vaqtINDUKTIVE : TIME := T#20s;
	tpT : ARRAY [1..10]  OF TP;
	ton1: TON;
	ton2 : TON;
	INDUK : ARRAY [1..5] OF INDUCTIVE;
	C16104_RDY_5: BOOL;
	C16104T_5: BOOL;
	C16104_SRT_5: BOOL;
	C16104_REM_5: BOOL;
	simul1: BOOL;
	X16106M1_REM_5: BOOL;
	X16106M1_SRT_TRIG: F_TRIGs;
	X16106M1_STP_TRIG: F_TRIGs;
	HJGJH: F_TRIGs;
	TOF1: TON;
	C16103_WRK_5: BOOL;
	L16003_SRT_G_5: BOOL;
	X16106M1_SRT_TRIG2: F_TRIGs;
	stopTEG_TP : TP;
END_VAR
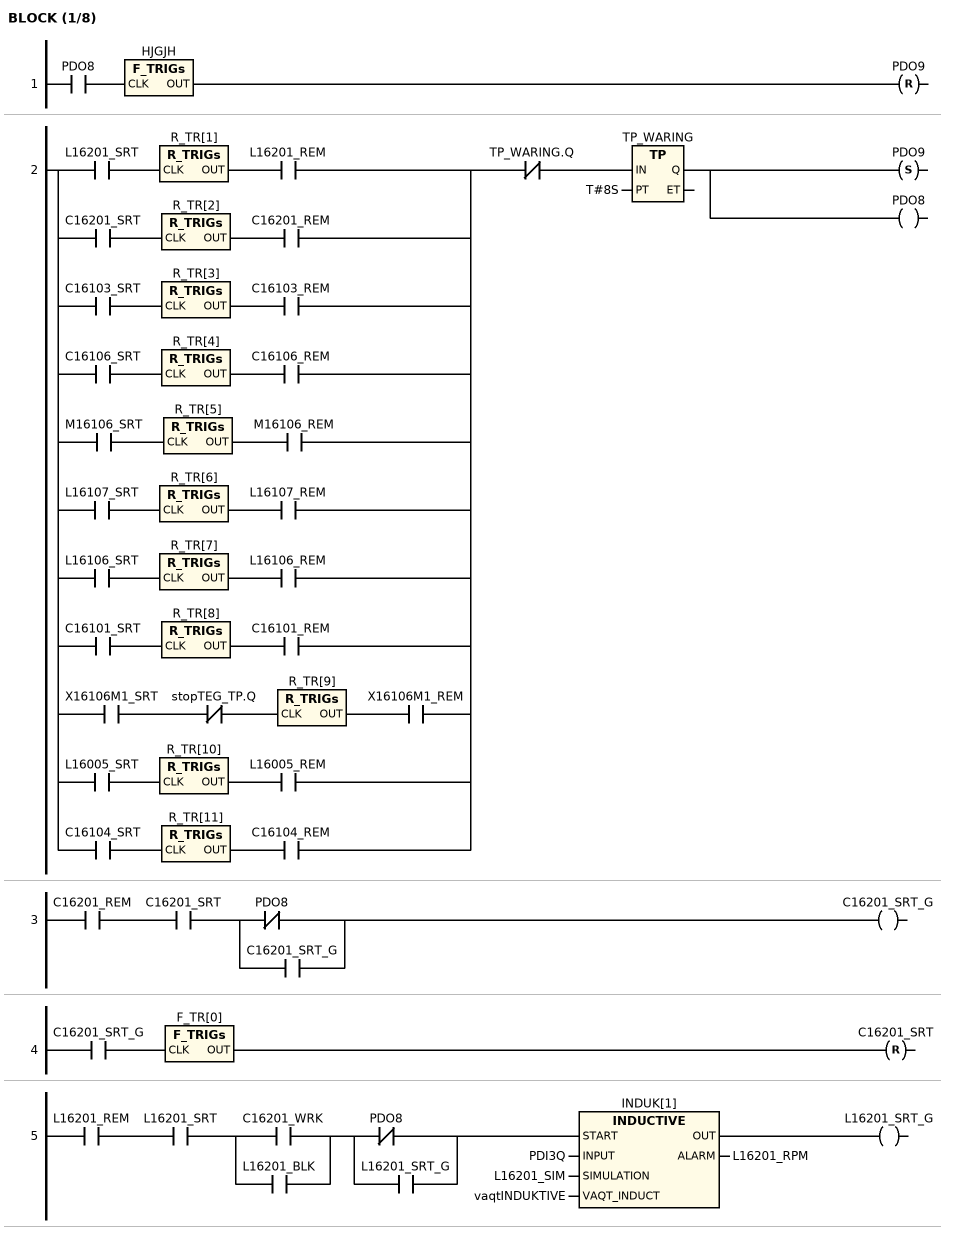
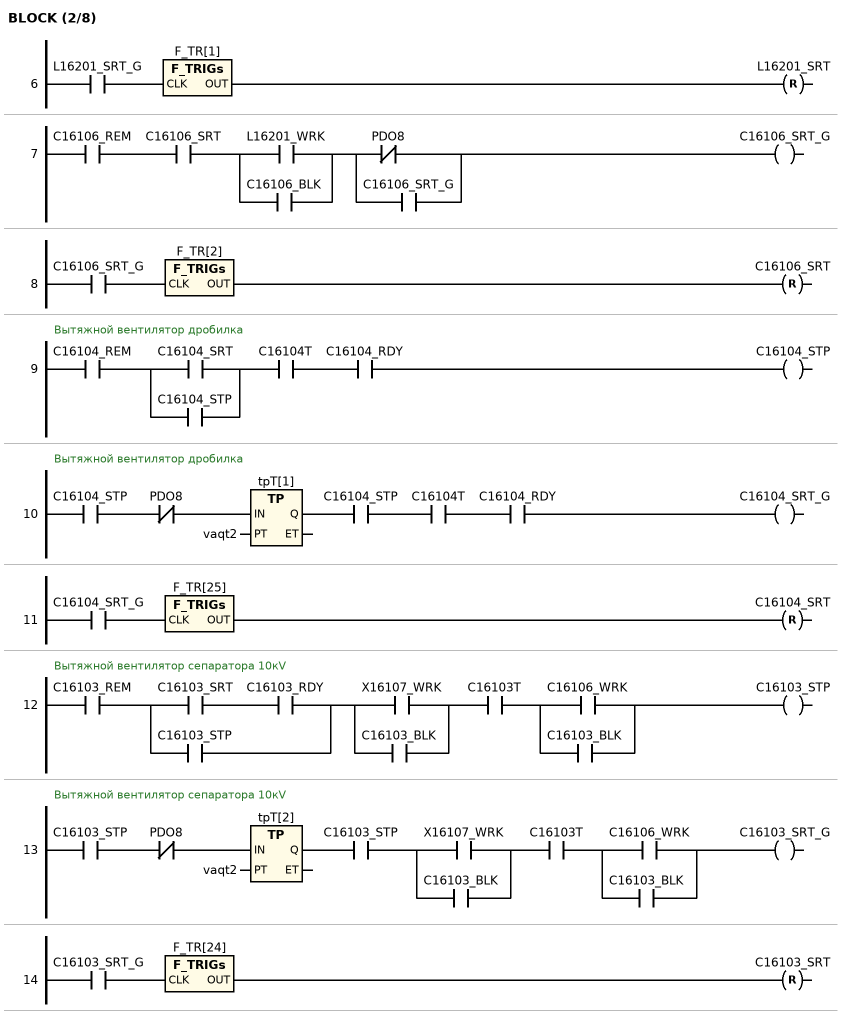
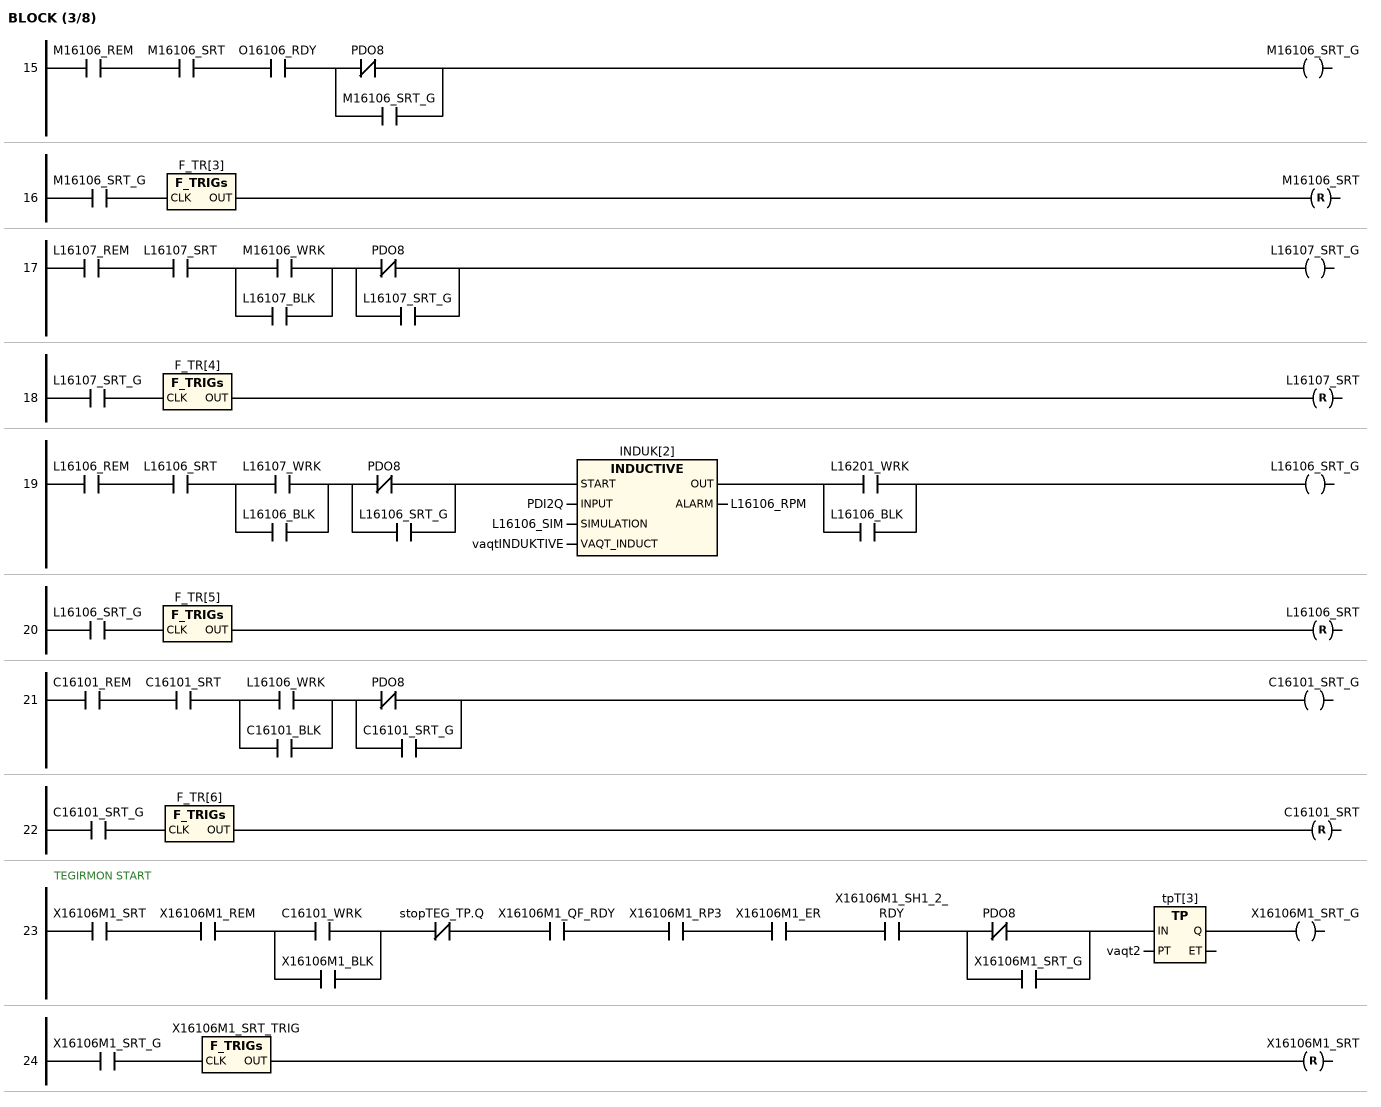
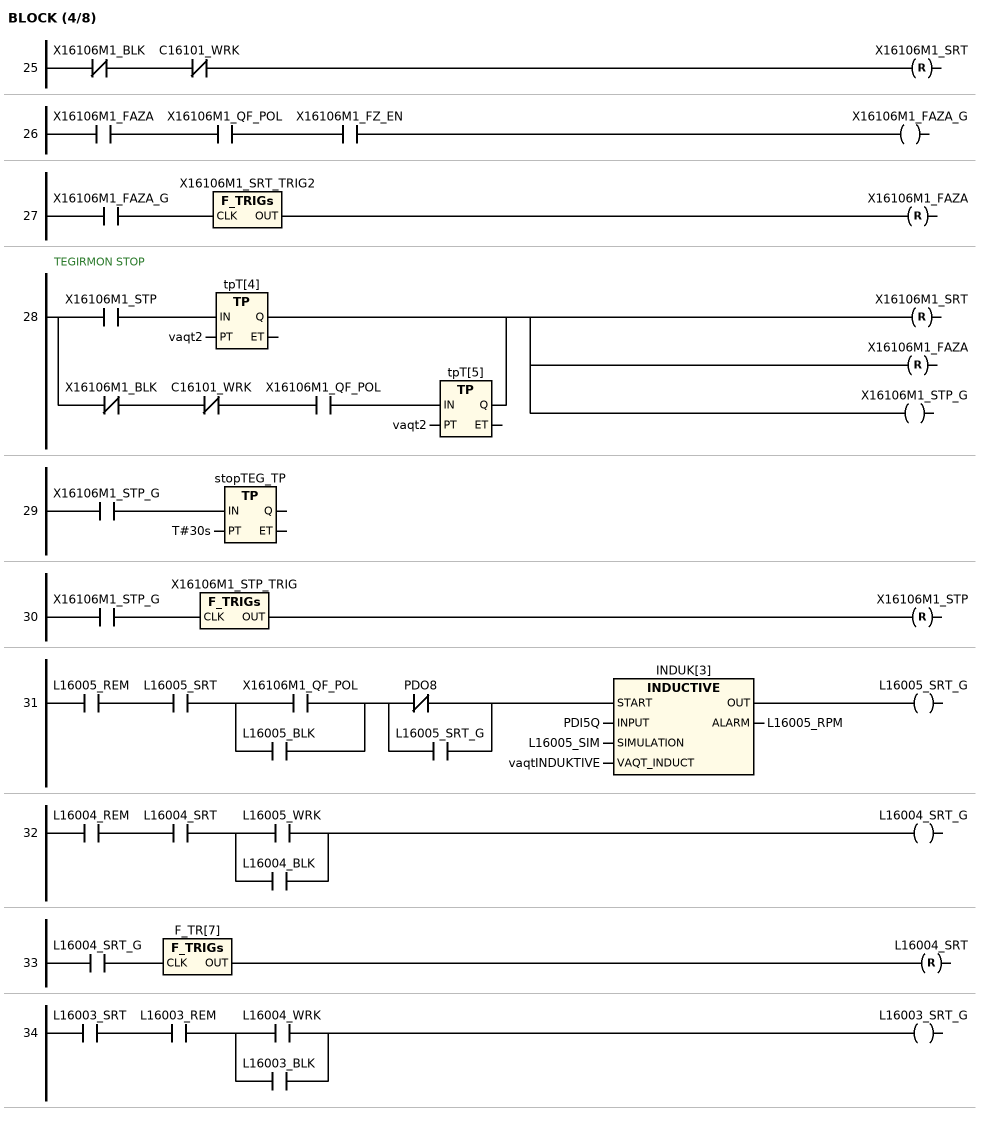
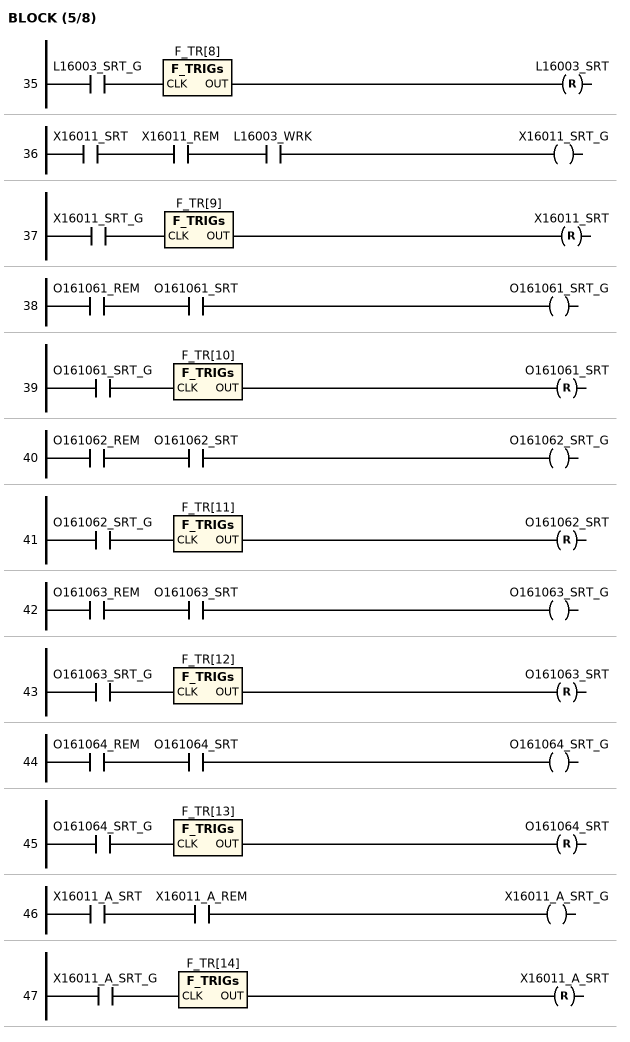
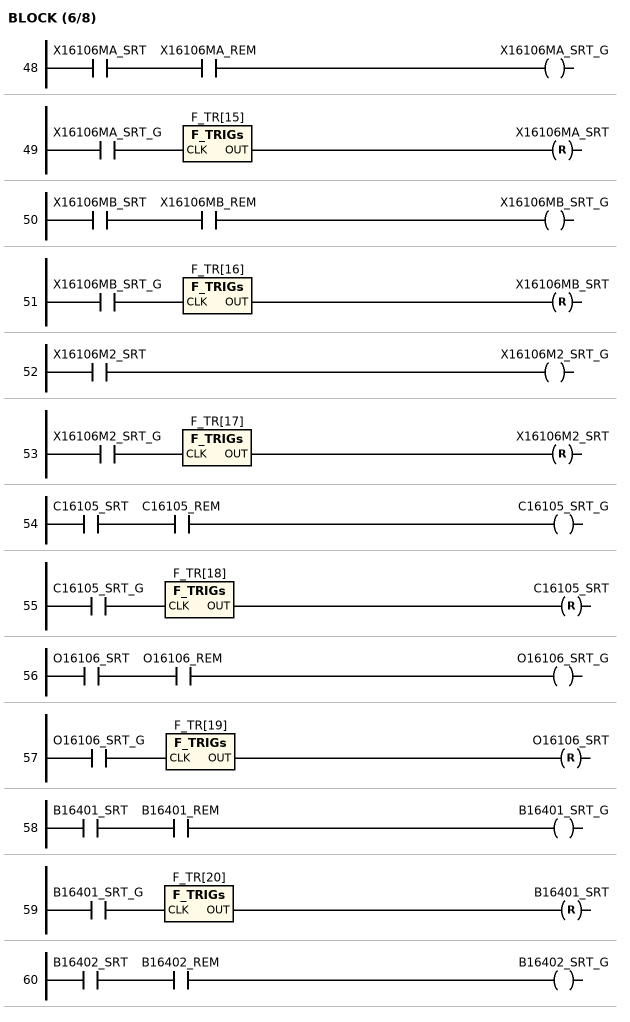
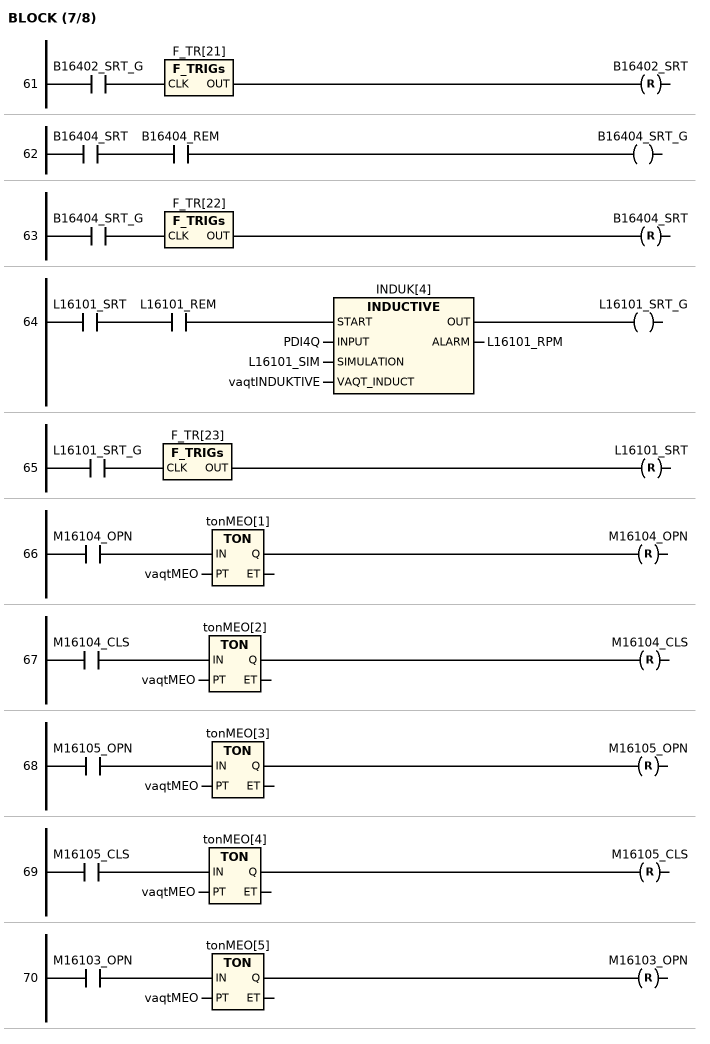
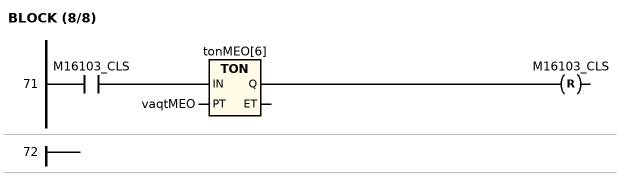
_LD_ (* Ladder Diagram *)
NETWORK 1
	[PDO8] - HJGJH:F_TRIGs(CLK: *) --- (R PDO9)
NETWORK 2
	{ [L16201_SRT] - R_TR[1]:R_TRIGs(CLK: *) - [L16201_REM] | [C16201_SRT] - R_TR[2]:R_TRIGs(CLK: *) - [C16201_REM] | [C16103_SRT] - R_TR[3]:R_TRIGs(CLK: *) - [C16103_REM] | [C16106_SRT] - R_TR[4]:R_TRIGs(CLK: *) - [C16106_REM] | [M16106_SRT] - R_TR[5]:R_TRIGs(CLK: *) - [M16106_REM] | [L16107_SRT] - R_TR[6]:R_TRIGs(CLK: *) - [L16107_REM] | [L16106_SRT] - R_TR[7]:R_TRIGs(CLK: *) - [L16106_REM] | [C16101_SRT] - R_TR[8]:R_TRIGs(CLK: *) - [C16101_REM] | [X16106M1_SRT] - [/stopTEG_TP.Q] - R_TR[9]:R_TRIGs(CLK: *) - [X16106M1_REM] | [L16005_SRT] - R_TR[10]:R_TRIGs(CLK: *) - [L16005_REM] | [C16104_SRT] - R_TR[11]:R_TRIGs(CLK: *) - [C16104_REM] } - [/TP_WARING.Q] - TP_WARING:TP(IN: *, PT: T#8S) --- (S PDO9) (PDO8)
NETWORK 3
	[C16201_REM] - [C16201_SRT] - { [/PDO8] | [C16201_SRT_G] } --- (C16201_SRT_G)
NETWORK 4
	[C16201_SRT_G] - F_TR[0]:F_TRIGs(CLK: *) --- (R C16201_SRT)
NETWORK 5
	[L16201_REM] - [L16201_SRT] - { [C16201_WRK] | [L16201_BLK] } - { [/PDO8] | [L16201_SRT_G] } - INDUK[1]:INDUCTIVE(START: *, INPUT: PDI3Q, SIMULATION: L16201_SIM, VAQT_INDUCT: vaqtINDUKTIVE, ALARM => L16201_RPM) --- (L16201_SRT_G)
NETWORK 6
	[L16201_SRT_G] - F_TR[1]:F_TRIGs(CLK: *) --- (R L16201_SRT)
NETWORK 7
	[C16106_REM] - [C16106_SRT] - { [L16201_WRK] | [C16106_BLK] } - { [/PDO8] | [C16106_SRT_G] } --- (C16106_SRT_G)
NETWORK 8
	[C16106_SRT_G] - F_TR[2]:F_TRIGs(CLK: *) --- (R C16106_SRT)
NETWORK 9 (* Вытяжной вентилятор дробилка *)
	[C16104_REM] - { [C16104_SRT] | [C16104_STP] } - [C16104T] - [C16104_RDY] --- (C16104_STP)
NETWORK 10 (* Вытяжной вентилятор дробилка *)
	[C16104_STP] - [/PDO8] - tpT[1]:TP(IN: *, PT: vaqt2) - [C16104_STP] - [C16104T] - [C16104_RDY] --- (C16104_SRT_G)
NETWORK 11
	[C16104_SRT_G] - F_TR[25]:F_TRIGs(CLK: *) --- (R C16104_SRT)
NETWORK 12 (* Вытяжной вентилятор сепаратора 10кV *)
	[C16103_REM] - { [C16103_SRT] - [C16103_RDY] | [C16103_STP] } - { [X16107_WRK] | [C16103_BLK] } - [C16103T] - { [C16106_WRK] | [C16103_BLK] } --- (C16103_STP)
NETWORK 13 (* Вытяжной вентилятор сепаратора 10кV *)
	[C16103_STP] - [/PDO8] - tpT[2]:TP(IN: *, PT: vaqt2) - [C16103_STP] - { [X16107_WRK] | [C16103_BLK] } - [C16103T] - { [C16106_WRK] | [C16103_BLK] } --- (C16103_SRT_G)
NETWORK 14
	[C16103_SRT_G] - F_TR[24]:F_TRIGs(CLK: *) --- (R C16103_SRT)
NETWORK 15
	[M16106_REM] - [M16106_SRT] - [O16106_RDY] - { [/PDO8] | [M16106_SRT_G] } --- (M16106_SRT_G)
NETWORK 16
	[M16106_SRT_G] - F_TR[3]:F_TRIGs(CLK: *) --- (R M16106_SRT)
NETWORK 17
	[L16107_REM] - [L16107_SRT] - { [M16106_WRK] | [L16107_BLK] } - { [/PDO8] | [L16107_SRT_G] } --- (L16107_SRT_G)
NETWORK 18
	[L16107_SRT_G] - F_TR[4]:F_TRIGs(CLK: *) --- (R L16107_SRT)
NETWORK 19
	[L16106_REM] - [L16106_SRT] - { [L16107_WRK] | [L16106_BLK] } - { [/PDO8] | [L16106_SRT_G] } - INDUK[2]:INDUCTIVE(START: *, INPUT: PDI2Q, SIMULATION: L16106_SIM, VAQT_INDUCT: vaqtINDUKTIVE, ALARM => L16106_RPM) - { [L16201_WRK] | [L16106_BLK] } --- (L16106_SRT_G)
NETWORK 20
	[L16106_SRT_G] - F_TR[5]:F_TRIGs(CLK: *) --- (R L16106_SRT)
NETWORK 21
	[C16101_REM] - [C16101_SRT] - { [L16106_WRK] | [C16101_BLK] } - { [/PDO8] | [C16101_SRT_G] } --- (C16101_SRT_G)
NETWORK 22
	[C16101_SRT_G] - F_TR[6]:F_TRIGs(CLK: *) --- (R C16101_SRT)
NETWORK 23 (* TEGIRMON START *)
	[X16106M1_SRT] - [X16106M1_REM] - { [C16101_WRK] | [X16106M1_BLK] } - [/stopTEG_TP.Q] - [X16106M1_QF_RDY] - [X16106M1_RP3] - [X16106M1_ER] - [X16106M1_SH1_2_RDY] - { [/PDO8] | [X16106M1_SRT_G] } - tpT[3]:TP(IN: *, PT: vaqt2) --- (X16106M1_SRT_G)
NETWORK 24
	[X16106M1_SRT_G] - X16106M1_SRT_TRIG:F_TRIGs(CLK: *) --- (R X16106M1_SRT)
NETWORK 25
	[/X16106M1_BLK] - [/C16101_WRK] --- (R X16106M1_SRT)
NETWORK 26
	[X16106M1_FAZA] - [X16106M1_QF_POL] - [X16106M1_FZ_EN] --- (X16106M1_FAZA_G)
NETWORK 27
	[X16106M1_FAZA_G] - X16106M1_SRT_TRIG2:F_TRIGs(CLK: *) --- (R X16106M1_FAZA)
NETWORK 28 (* TEGIRMON STOP *)
	{ [X16106M1_STP] - tpT[4]:TP(IN: *, PT: vaqt2) | [/X16106M1_BLK] - [/C16101_WRK] - [X16106M1_QF_POL] - tpT[5]:TP(IN: *, PT: vaqt2) } --- (R X16106M1_SRT) (R X16106M1_FAZA) (X16106M1_STP_G)
NETWORK 29
	[X16106M1_STP_G] - stopTEG_TP:TP(IN: *, PT: T#30s)
NETWORK 30
	[X16106M1_STP_G] - X16106M1_STP_TRIG:F_TRIGs(CLK: *) --- (R X16106M1_STP)
NETWORK 31
	[L16005_REM] - [L16005_SRT] - { [X16106M1_QF_POL] | [L16005_BLK] } - { [/PDO8] | [L16005_SRT_G] } - INDUK[3]:INDUCTIVE(START: *, INPUT: PDI5Q, SIMULATION: L16005_SIM, VAQT_INDUCT: vaqtINDUKTIVE, ALARM => L16005_RPM) --- (L16005_SRT_G)
NETWORK 32
	[L16004_REM] - [L16004_SRT] - { [L16005_WRK] | [L16004_BLK] } --- (L16004_SRT_G)
NETWORK 33
	[L16004_SRT_G] - F_TR[7]:F_TRIGs(CLK: *) --- (R L16004_SRT)
NETWORK 34
	[L16003_SRT] - [L16003_REM] - { [L16004_WRK] | [L16003_BLK] } --- (L16003_SRT_G)
NETWORK 35
	[L16003_SRT_G] - F_TR[8]:F_TRIGs(CLK: *) --- (R L16003_SRT)
NETWORK 36
	[X16011_SRT] - [X16011_REM] - [L16003_WRK] --- (X16011_SRT_G)
NETWORK 37
	[X16011_SRT_G] - F_TR[9]:F_TRIGs(CLK: *) --- (R X16011_SRT)
NETWORK 38
	[O161061_REM] - [O161061_SRT] --- (O161061_SRT_G)
NETWORK 39
	[O161061_SRT_G] - F_TR[10]:F_TRIGs(CLK: *) --- (R O161061_SRT)
NETWORK 40
	[O161062_REM] - [O161062_SRT] --- (O161062_SRT_G)
NETWORK 41
	[O161062_SRT_G] - F_TR[11]:F_TRIGs(CLK: *) --- (R O161062_SRT)
NETWORK 42
	[O161063_REM] - [O161063_SRT] --- (O161063_SRT_G)
NETWORK 43
	[O161063_SRT_G] - F_TR[12]:F_TRIGs(CLK: *) --- (R O161063_SRT)
NETWORK 44
	[O161064_REM] - [O161064_SRT] --- (O161064_SRT_G)
NETWORK 45
	[O161064_SRT_G] - F_TR[13]:F_TRIGs(CLK: *) --- (R O161064_SRT)
NETWORK 46
	[X16011_A_SRT] - [X16011_A_REM] --- (X16011_A_SRT_G)
NETWORK 47
	[X16011_A_SRT_G] - F_TR[14]:F_TRIGs(CLK: *) --- (R X16011_A_SRT)
NETWORK 48
	[X16106MA_SRT] - [X16106MA_REM] --- (X16106MA_SRT_G)
NETWORK 49
	[X16106MA_SRT_G] - F_TR[15]:F_TRIGs(CLK: *) --- (R X16106MA_SRT)
NETWORK 50
	[X16106MB_SRT] - [X16106MB_REM] --- (X16106MB_SRT_G)
NETWORK 51
	[X16106MB_SRT_G] - F_TR[16]:F_TRIGs(CLK: *) --- (R X16106MB_SRT)
NETWORK 52
	[X16106M2_SRT] --- (X16106M2_SRT_G)
NETWORK 53
	[X16106M2_SRT_G] - F_TR[17]:F_TRIGs(CLK: *) --- (R X16106M2_SRT)
NETWORK 54
	[C16105_SRT] - [C16105_REM] --- (C16105_SRT_G)
NETWORK 55
	[C16105_SRT_G] - F_TR[18]:F_TRIGs(CLK: *) --- (R C16105_SRT)
NETWORK 56
	[O16106_SRT] - [O16106_REM] --- (O16106_SRT_G)
NETWORK 57
	[O16106_SRT_G] - F_TR[19]:F_TRIGs(CLK: *) --- (R O16106_SRT)
NETWORK 58
	[B16401_SRT] - [B16401_REM] --- (B16401_SRT_G)
NETWORK 59
	[B16401_SRT_G] - F_TR[20]:F_TRIGs(CLK: *) --- (R B16401_SRT)
NETWORK 60
	[B16402_SRT] - [B16402_REM] --- (B16402_SRT_G)
NETWORK 61
	[B16402_SRT_G] - F_TR[21]:F_TRIGs(CLK: *) --- (R B16402_SRT)
NETWORK 62
	[B16404_SRT] - [B16404_REM] --- (B16404_SRT_G)
NETWORK 63
	[B16404_SRT_G] - F_TR[22]:F_TRIGs(CLK: *) --- (R B16404_SRT)
NETWORK 64
	[L16101_SRT] - [L16101_REM] - INDUK[4]:INDUCTIVE(START: *, INPUT: PDI4Q, SIMULATION: L16101_SIM, VAQT_INDUCT: vaqtINDUKTIVE, ALARM => L16101_RPM) --- (L16101_SRT_G)
NETWORK 65
	[L16101_SRT_G] - F_TR[23]:F_TRIGs(CLK: *) --- (R L16101_SRT)
NETWORK 66
	[M16104_OPN] - tonMEO[1]:TON(IN: *, PT: vaqtMEO) --- (R M16104_OPN)
NETWORK 67
	[M16104_CLS] - tonMEO[2]:TON(IN: *, PT: vaqtMEO) --- (R M16104_CLS)
NETWORK 68
	[M16105_OPN] - tonMEO[3]:TON(IN: *, PT: vaqtMEO) --- (R M16105_OPN)
NETWORK 69
	[M16105_CLS] - tonMEO[4]:TON(IN: *, PT: vaqtMEO) --- (R M16105_CLS)
NETWORK 70
	[M16103_OPN] - tonMEO[5]:TON(IN: *, PT: vaqtMEO) --- (R M16103_OPN)
NETWORK 71
	[M16103_CLS] - tonMEO[6]:TON(IN: *, PT: vaqtMEO) --- (R M16103_CLS)
NETWORK 72
	*
_END_LD_
(* the same logic as Structured Text *)
(* Network 1 *)
HJGJH(CLK := PDO8);
IF HJGJH.OUT THEN PDO9 := FALSE; END_IF;
(* Network 2 *)
R_TR[1](CLK := L16201_SRT);
R_TR[2](CLK := C16201_SRT);
R_TR[3](CLK := C16103_SRT);
R_TR[4](CLK := C16106_SRT);
R_TR[5](CLK := M16106_SRT);
R_TR[6](CLK := L16107_SRT);
R_TR[7](CLK := L16106_SRT);
R_TR[8](CLK := C16101_SRT);
R_TR[9](CLK := X16106M1_SRT AND NOT stopTEG_TP.Q);
R_TR[10](CLK := L16005_SRT);
R_TR[11](CLK := C16104_SRT);
TP_WARING(IN := (R_TR[1].OUT AND L16201_REM OR R_TR[2].OUT AND C16201_REM OR R_TR[3].OUT AND C16103_REM OR R_TR[4].OUT AND C16106_REM OR R_TR[5].OUT AND M16106_REM OR R_TR[6].OUT AND L16107_REM OR R_TR[7].OUT AND L16106_REM OR R_TR[8].OUT AND C16101_REM OR R_TR[9].OUT AND X16106M1_REM OR R_TR[10].OUT AND L16005_REM OR R_TR[11].OUT AND C16104_REM) AND NOT TP_WARING.Q, PT := T#8S);
IF TP_WARING.Q THEN PDO9 := TRUE; END_IF;
PDO8 := TP_WARING.Q;
(* Network 3 *)
C16201_SRT_G := C16201_REM AND C16201_SRT AND (NOT PDO8 OR C16201_SRT_G);
(* Network 4 *)
F_TR[0](CLK := C16201_SRT_G);
IF F_TR[0].OUT THEN C16201_SRT := FALSE; END_IF;
(* Network 5 *)
INDUK[1](START := L16201_REM AND L16201_SRT AND (C16201_WRK OR L16201_BLK) AND (NOT PDO8 OR L16201_SRT_G), INPUT := PDI3Q, SIMULATION := L16201_SIM, VAQT_INDUCT := vaqtINDUKTIVE);
L16201_RPM := INDUK[1].ALARM;
L16201_SRT_G := INDUK[1].OUT;
(* Network 6 *)
F_TR[1](CLK := L16201_SRT_G);
IF F_TR[1].OUT THEN L16201_SRT := FALSE; END_IF;
(* Network 7 *)
C16106_SRT_G := C16106_REM AND C16106_SRT AND (L16201_WRK OR C16106_BLK) AND (NOT PDO8 OR C16106_SRT_G);
(* Network 8 *)
F_TR[2](CLK := C16106_SRT_G);
IF F_TR[2].OUT THEN C16106_SRT := FALSE; END_IF;
(* Network 9: Вытяжной вентилятор дробилка *)
C16104_STP := C16104_REM AND (C16104_SRT OR C16104_STP) AND C16104T AND C16104_RDY;
(* Network 10: Вытяжной вентилятор дробилка *)
tpT[1](IN := C16104_STP AND NOT PDO8, PT := vaqt2);
C16104_SRT_G := tpT[1].Q AND C16104_STP AND C16104T AND C16104_RDY;
(* Network 11 *)
F_TR[25](CLK := C16104_SRT_G);
IF F_TR[25].OUT THEN C16104_SRT := FALSE; END_IF;
(* Network 12: Вытяжной вентилятор сепаратора 10кV *)
C16103_STP := C16103_REM AND (C16103_SRT AND C16103_RDY OR C16103_STP) AND (X16107_WRK OR C16103_BLK) AND C16103T AND (C16106_WRK OR C16103_BLK);
(* Network 13: Вытяжной вентилятор сепаратора 10кV *)
tpT[2](IN := C16103_STP AND NOT PDO8, PT := vaqt2);
C16103_SRT_G := tpT[2].Q AND C16103_STP AND (X16107_WRK OR C16103_BLK) AND C16103T AND (C16106_WRK OR C16103_BLK);
(* Network 14 *)
F_TR[24](CLK := C16103_SRT_G);
IF F_TR[24].OUT THEN C16103_SRT := FALSE; END_IF;
(* Network 15 *)
M16106_SRT_G := M16106_REM AND M16106_SRT AND O16106_RDY AND (NOT PDO8 OR M16106_SRT_G);
(* Network 16 *)
F_TR[3](CLK := M16106_SRT_G);
IF F_TR[3].OUT THEN M16106_SRT := FALSE; END_IF;
(* Network 17 *)
L16107_SRT_G := L16107_REM AND L16107_SRT AND (M16106_WRK OR L16107_BLK) AND (NOT PDO8 OR L16107_SRT_G);
(* Network 18 *)
F_TR[4](CLK := L16107_SRT_G);
IF F_TR[4].OUT THEN L16107_SRT := FALSE; END_IF;
(* Network 19 *)
INDUK[2](START := L16106_REM AND L16106_SRT AND (L16107_WRK OR L16106_BLK) AND (NOT PDO8 OR L16106_SRT_G), INPUT := PDI2Q, SIMULATION := L16106_SIM, VAQT_INDUCT := vaqtINDUKTIVE);
L16106_RPM := INDUK[2].ALARM;
L16106_SRT_G := INDUK[2].OUT AND (L16201_WRK OR L16106_BLK);
(* Network 20 *)
F_TR[5](CLK := L16106_SRT_G);
IF F_TR[5].OUT THEN L16106_SRT := FALSE; END_IF;
(* Network 21 *)
C16101_SRT_G := C16101_REM AND C16101_SRT AND (L16106_WRK OR C16101_BLK) AND (NOT PDO8 OR C16101_SRT_G);
(* Network 22 *)
F_TR[6](CLK := C16101_SRT_G);
IF F_TR[6].OUT THEN C16101_SRT := FALSE; END_IF;
(* Network 23: TEGIRMON START *)
tpT[3](IN := X16106M1_SRT AND X16106M1_REM AND (C16101_WRK OR X16106M1_BLK) AND NOT stopTEG_TP.Q AND X16106M1_QF_RDY AND X16106M1_RP3 AND X16106M1_ER AND X16106M1_SH1_2_RDY AND (NOT PDO8 OR X16106M1_SRT_G), PT := vaqt2);
X16106M1_SRT_G := tpT[3].Q;
(* Network 24 *)
X16106M1_SRT_TRIG(CLK := X16106M1_SRT_G);
IF X16106M1_SRT_TRIG.OUT THEN X16106M1_SRT := FALSE; END_IF;
(* Network 25 *)
IF NOT X16106M1_BLK AND NOT C16101_WRK THEN X16106M1_SRT := FALSE; END_IF;
(* Network 26 *)
X16106M1_FAZA_G := X16106M1_FAZA AND X16106M1_QF_POL AND X16106M1_FZ_EN;
(* Network 27 *)
X16106M1_SRT_TRIG2(CLK := X16106M1_FAZA_G);
IF X16106M1_SRT_TRIG2.OUT THEN X16106M1_FAZA := FALSE; END_IF;
(* Network 28: TEGIRMON STOP *)
tpT[4](IN := X16106M1_STP, PT := vaqt2);
tpT[5](IN := NOT X16106M1_BLK AND NOT C16101_WRK AND X16106M1_QF_POL, PT := vaqt2);
IF tpT[4].Q OR tpT[5].Q THEN X16106M1_SRT := FALSE; END_IF;
IF tpT[4].Q OR tpT[5].Q THEN X16106M1_FAZA := FALSE; END_IF;
X16106M1_STP_G := tpT[4].Q OR tpT[5].Q;
(* Network 29 *)
stopTEG_TP(IN := X16106M1_STP_G, PT := T#30s);
(* Network 30 *)
X16106M1_STP_TRIG(CLK := X16106M1_STP_G);
IF X16106M1_STP_TRIG.OUT THEN X16106M1_STP := FALSE; END_IF;
(* Network 31 *)
INDUK[3](START := L16005_REM AND L16005_SRT AND (X16106M1_QF_POL OR L16005_BLK) AND (NOT PDO8 OR L16005_SRT_G), INPUT := PDI5Q, SIMULATION := L16005_SIM, VAQT_INDUCT := vaqtINDUKTIVE);
L16005_RPM := INDUK[3].ALARM;
L16005_SRT_G := INDUK[3].OUT;
(* Network 32 *)
L16004_SRT_G := L16004_REM AND L16004_SRT AND (L16005_WRK OR L16004_BLK);
(* Network 33 *)
F_TR[7](CLK := L16004_SRT_G);
IF F_TR[7].OUT THEN L16004_SRT := FALSE; END_IF;
(* Network 34 *)
L16003_SRT_G := L16003_SRT AND L16003_REM AND (L16004_WRK OR L16003_BLK);
(* Network 35 *)
F_TR[8](CLK := L16003_SRT_G);
IF F_TR[8].OUT THEN L16003_SRT := FALSE; END_IF;
(* Network 36 *)
X16011_SRT_G := X16011_SRT AND X16011_REM AND L16003_WRK;
(* Network 37 *)
F_TR[9](CLK := X16011_SRT_G);
IF F_TR[9].OUT THEN X16011_SRT := FALSE; END_IF;
(* Network 38 *)
O161061_SRT_G := O161061_REM AND O161061_SRT;
(* Network 39 *)
F_TR[10](CLK := O161061_SRT_G);
IF F_TR[10].OUT THEN O161061_SRT := FALSE; END_IF;
(* Network 40 *)
O161062_SRT_G := O161062_REM AND O161062_SRT;
(* Network 41 *)
F_TR[11](CLK := O161062_SRT_G);
IF F_TR[11].OUT THEN O161062_SRT := FALSE; END_IF;
(* Network 42 *)
O161063_SRT_G := O161063_REM AND O161063_SRT;
(* Network 43 *)
F_TR[12](CLK := O161063_SRT_G);
IF F_TR[12].OUT THEN O161063_SRT := FALSE; END_IF;
(* Network 44 *)
O161064_SRT_G := O161064_REM AND O161064_SRT;
(* Network 45 *)
F_TR[13](CLK := O161064_SRT_G);
IF F_TR[13].OUT THEN O161064_SRT := FALSE; END_IF;
(* Network 46 *)
X16011_A_SRT_G := X16011_A_SRT AND X16011_A_REM;
(* Network 47 *)
F_TR[14](CLK := X16011_A_SRT_G);
IF F_TR[14].OUT THEN X16011_A_SRT := FALSE; END_IF;
(* Network 48 *)
X16106MA_SRT_G := X16106MA_SRT AND X16106MA_REM;
(* Network 49 *)
F_TR[15](CLK := X16106MA_SRT_G);
IF F_TR[15].OUT THEN X16106MA_SRT := FALSE; END_IF;
(* Network 50 *)
X16106MB_SRT_G := X16106MB_SRT AND X16106MB_REM;
(* Network 51 *)
F_TR[16](CLK := X16106MB_SRT_G);
IF F_TR[16].OUT THEN X16106MB_SRT := FALSE; END_IF;
(* Network 52 *)
X16106M2_SRT_G := X16106M2_SRT;
(* Network 53 *)
F_TR[17](CLK := X16106M2_SRT_G);
IF F_TR[17].OUT THEN X16106M2_SRT := FALSE; END_IF;
(* Network 54 *)
C16105_SRT_G := C16105_SRT AND C16105_REM;
(* Network 55 *)
F_TR[18](CLK := C16105_SRT_G);
IF F_TR[18].OUT THEN C16105_SRT := FALSE; END_IF;
(* Network 56 *)
O16106_SRT_G := O16106_SRT AND O16106_REM;
(* Network 57 *)
F_TR[19](CLK := O16106_SRT_G);
IF F_TR[19].OUT THEN O16106_SRT := FALSE; END_IF;
(* Network 58 *)
B16401_SRT_G := B16401_SRT AND B16401_REM;
(* Network 59 *)
F_TR[20](CLK := B16401_SRT_G);
IF F_TR[20].OUT THEN B16401_SRT := FALSE; END_IF;
(* Network 60 *)
B16402_SRT_G := B16402_SRT AND B16402_REM;
(* Network 61 *)
F_TR[21](CLK := B16402_SRT_G);
IF F_TR[21].OUT THEN B16402_SRT := FALSE; END_IF;
(* Network 62 *)
B16404_SRT_G := B16404_SRT AND B16404_REM;
(* Network 63 *)
F_TR[22](CLK := B16404_SRT_G);
IF F_TR[22].OUT THEN B16404_SRT := FALSE; END_IF;
(* Network 64 *)
INDUK[4](START := L16101_SRT AND L16101_REM, INPUT := PDI4Q, SIMULATION := L16101_SIM, VAQT_INDUCT := vaqtINDUKTIVE);
L16101_RPM := INDUK[4].ALARM;
L16101_SRT_G := INDUK[4].OUT;
(* Network 65 *)
F_TR[23](CLK := L16101_SRT_G);
IF F_TR[23].OUT THEN L16101_SRT := FALSE; END_IF;
(* Network 66 *)
tonMEO[1](IN := M16104_OPN, PT := vaqtMEO);
IF tonMEO[1].Q THEN M16104_OPN := FALSE; END_IF;
(* Network 67 *)
tonMEO[2](IN := M16104_CLS, PT := vaqtMEO);
IF tonMEO[2].Q THEN M16104_CLS := FALSE; END_IF;
(* Network 68 *)
tonMEO[3](IN := M16105_OPN, PT := vaqtMEO);
IF tonMEO[3].Q THEN M16105_OPN := FALSE; END_IF;
(* Network 69 *)
tonMEO[4](IN := M16105_CLS, PT := vaqtMEO);
IF tonMEO[4].Q THEN M16105_CLS := FALSE; END_IF;
(* Network 70 *)
tonMEO[5](IN := M16103_OPN, PT := vaqtMEO);
IF tonMEO[5].Q THEN M16103_OPN := FALSE; END_IF;
(* Network 71 *)
tonMEO[6](IN := M16103_CLS, PT := vaqtMEO);
IF tonMEO[6].Q THEN M16103_CLS := FALSE; END_IF;
(* Network 72 *)
END_PROGRAM

(* POU R_TRIGs, LD *)
FUNCTION_BLOCK R_TRIGs
VAR_INPUT
	CLK : BOOL;
END_VAR
VAR_OUTPUT
	OUT : BOOL;
END_VAR
VAR
	TMP: BOOL;
	tp1: TP;
END_VAR
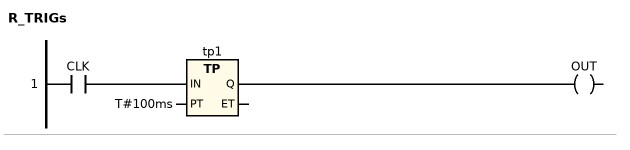
_LD_ (* Ladder Diagram *)
NETWORK 1
	[CLK] - tp1:TP(IN: *, PT: T#100ms) --- (OUT)
_END_LD_
(* the same logic as Structured Text *)
(* Network 1 *)
tp1(IN := CLK, PT := T#100ms);
OUT := tp1.Q;
END_FUNCTION_BLOCK

(* POU F_TRIGs, CFC *)
FUNCTION_BLOCK F_TRIGs
VAR_INPUT
	CLK : BOOL;

END_VAR
VAR_OUTPUT
	OUT : BOOL;
END_VAR
VAR
	VAQT : TIME := T#500ms;
	Ton1: TON;
END_VAR
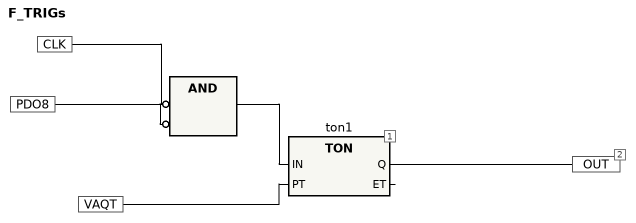
_CFC_ (* Continuous Function Chart, elements in execution order *)
#0 AND(NOT CLK, NOT PDO8)
#1 ton1:TON(IN: #0, PT: VAQT)
#2 OUT <= #1.Q
_END_CFC_
(* the same logic as Structured Text *)
ton1(IN := NOT CLK AND NOT PDO8, PT := VAQT);
OUT := ton1.Q;
END_FUNCTION_BLOCK

(* POU vaqt, ST *)
PROGRAM vaqt
(*o'zgaruvchilarni e'lon qilish*)
VAR
	tmr, tmr2, tmr_f, tmr_sr : TON;
	sum_mV : REAL;
	old_weight_tr : REAL;
	sum_cnt : INT;
	filtr_mV : REAL;
	sr_proiz : REAL;
	sr_cnt : INT;
	sr_speed : REAL;
	GetTime: CurTimeEx;
	TDate: SystemTimeDate;
	Sys_Time: SysTime64;
	need_day : UINT;
	mb_count_month: WORD;
	mb_count_old_month: WORD;
	mb_count_smena: WORD;
	mb_count_old_smena: WORD;
	mb_count_soat_tch: WORD;
	mb_count_old_soat_tch: WORD;



END_VAR
(*o'zgaruvchilarni e'lon qilish*)
TDate.Day :=0;
TDate.DayOfWeek :=0;
TDate.dwHighMsec :=0;
TDate.dwLowMSecs :=0;
TDate.Milliseconds :=0;
TDate.Minute :=0;
TDate.Second :=0;
TDate.Hour :=0;
TDate.Year :=0;
TDate.Month :=0;
Sys_time.ulHigh :=0;
Sys_time.ulLow :=0;
GetTime (SystemTime:=Sys_Time , TimeDate:= TDate);

CASE TDate.Month OF
	1, 3, 5, 7, 8, 10, 12 : need_day := 31; (*Agar 1, 3, .. 12 oy lar bulsa 31 kuni hisoblagichni nol qilish*)
	2 : IF (TDate.Year MOD 4  = 0 AND TDate.Year MOD 100 > 0 OR TDate.Year MOD 400 = 0) THEN
			need_day := 29;  (*Agar yil kabisa yili  bulsa 29 kuni hisoblagichni nol qilish*)
		ELSE
			need_day := 28;  (*Agar yil kabisa yili EMAS bulsa 29 kuni hisoblagichni nol qilish*)
		END_IF;
	4, 6, 9, 11 : need_day := 30; (*Qolgan oylarda 30 kuni nol qilish*)
END_CASE;


(*==========================================================*)
(* bir smenalik tonnani boshqa registrga yozib qo'yish*)
IF(TDate.Minute = 59) AND(TDate.Second = 59) AND (TDate.Hour = 23) OR SYNC THEN
	(*mb_count_old_smena := mb_count_smena;*)
	eski_counter_1 := counter_1;
	eski_counter_2 := counter_2;
	eski_counter_3 := counter_3;
	eski_counter_4 := counter_4;
	SYNC := FALSE;

END_IF;
(*
count_hour1 := DWORD_TO_WORD(counter_1 - eski_counter_1);
count_hour2 := DWORD_TO_WORD(counter_2 - eski_counter_2);
count_hour3 := DWORD_TO_WORD(counter_3 - eski_counter_3);
count_hour4 := DWORD_TO_WORD(counter_4 - eski_counter_4);
*)
count_hour1 := REAL_TO_WORD (counter_1 - eski_counter_1);
count_hour2 := REAL_TO_WORD(counter_2 - eski_counter_2);
count_hour3 := REAL_TO_WORD(counter_3 - eski_counter_3);
count_hour4 := REAL_TO_WORD(counter_4 - eski_counter_4);

count_TOTAL := count_hour1 + count_hour2 + count_hour3 + count_hour4;





















(*==========================*)

(*tok_chast := 4+(mmb_speed := (chast * 6.76)/10000;b_percent_chast * 0.16);*
mb_speed := (chast * 6.76)/10000;



tmr(in := TRUE, pt := T#1s);
IF (tmr.Q = FALSE) THEN
	sum_cnt := sum_cnt + 1;
	sum_mV := sum_mV / sum_cnt + mV_7016;
ELSE
	filtr_mV := mV_7016;
	sum_mV := 0;
	sum_cnt := 1;
	tmr(in := FALSE);
END_IF;
*)
END_PROGRAM

(* POU INDUCTIVE, CFC *)
FUNCTION_BLOCK INDUCTIVE
VAR_INPUT
	START : BOOL;
	INPUT : BOOL;
	SIMULATION : BOOL := FALSE;
	VAQT_INDUCT : TIME := T#20S;
END_VAR
VAR_OUTPUT
	OUT : BOOL;
	ALARM : BOOL;
END_VAR
VAR
	TON1: TON;
	TON2: TON;
	TON3: TON;
	RUNNING : BOOL;
END_VAR
VAR (* helpers for the ST form of the networks *)
	_t11 : BOOL;
	_t12 : BOOL;
	_t7 : BOOL;
	_t31 : BOOL;
	_t18 : BOOL;
END_VAR
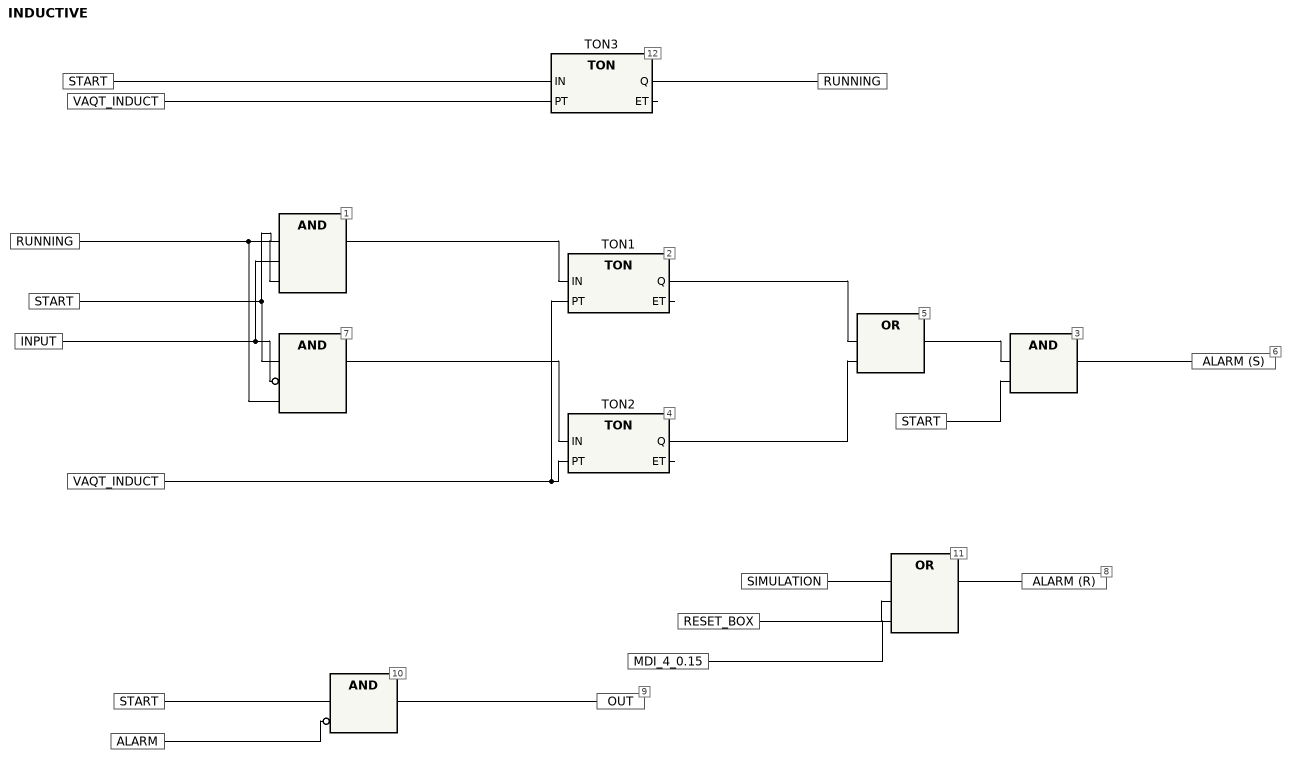
_CFC_ (* Continuous Function Chart, elements in execution order *)
#0 RUNNING <= #12.Q
#1 AND(START, INPUT, RUNNING)
#2 TON1:TON(IN: #1, PT: VAQT_INDUCT)
#3 AND(#5, START)
#4 TON2:TON(IN: #7, PT: VAQT_INDUCT)
#5 OR(#2.Q, #4.Q)
#6 S ALARM <= #3
#7 AND(START, NOT INPUT, RUNNING)
#8 R ALARM <= #11
#9 OUT <= #10
#10 AND(START, NOT ALARM)
#11 OR(SIMULATION, RESET_BOX, MDI_4_0.15)
#12 TON3:TON(IN: START, PT: VAQT_INDUCT)
_END_CFC_
(* the same logic as Structured Text *)
RUNNING := TON3.Q;
TON1(IN := START AND INPUT AND RUNNING, PT := VAQT_INDUCT);
_t12 := _t11 AND START;
TON2(IN := _t7, PT := VAQT_INDUCT);
_t11 := TON1.Q OR TON2.Q;
IF _t12 THEN ALARM := TRUE; END_IF;
_t7 := START AND NOT INPUT AND RUNNING;
IF _t31 THEN ALARM := FALSE; END_IF;
OUT := _t18;
_t18 := START AND NOT ALARM;
_t31 := SIMULATION OR RESET_BOX OR MDI_4_0.15;
TON3(IN := START, PT := VAQT_INDUCT);
END_FUNCTION_BLOCK

(* POU ALARM_RPM, CFC *)
PROGRAM ALARM_RPM
VAR
	RTRIG : ARRAY [1..16] OF R_TRIGs;
	VAQT : TIME := T#100MS;
	ind : ARRAY[1..3]  OF INDUCTIVE;
END_VAR
VAR (* helpers for the ST form of the networks *)
	_t46 : BOOL;
END_VAR
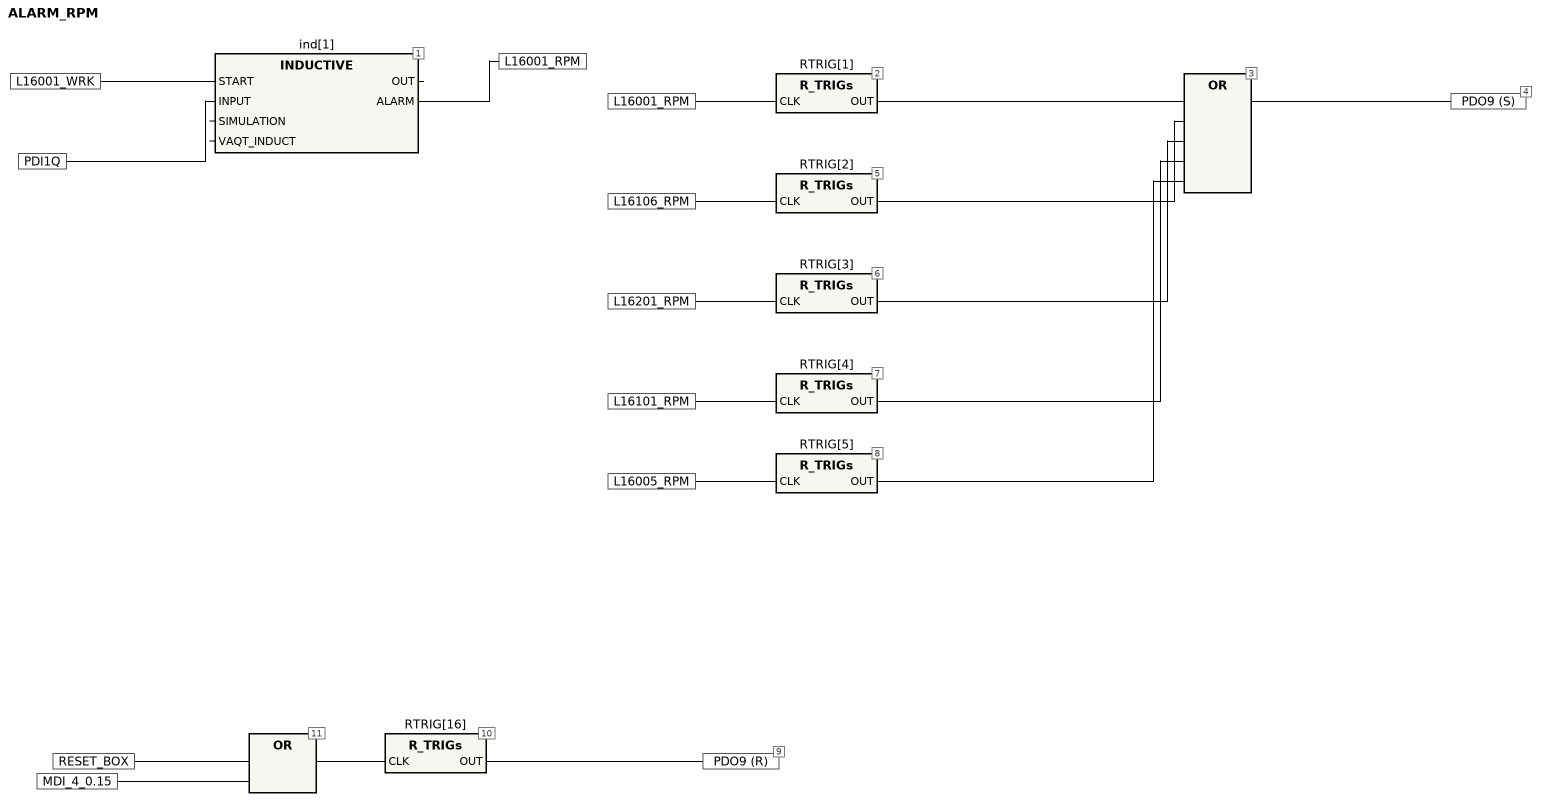
_CFC_ (* Continuous Function Chart, elements in execution order *)
#0 L16001_RPM <= #1.ALARM
#1 ind[1]:INDUCTIVE(START: L16001_WRK, INPUT: PDI1Q, SIMULATION: -, VAQT_INDUCT: -)
#2 RTRIG[1]:R_TRIGs(CLK: L16001_RPM)
#3 OR(#2.OUT, #5.OUT, #6.OUT, #7.OUT, #8.OUT)
#4 S PDO9 <= #3
#5 RTRIG[2]:R_TRIGs(CLK: L16106_RPM)
#6 RTRIG[3]:R_TRIGs(CLK: L16201_RPM)
#7 RTRIG[4]:R_TRIGs(CLK: L16101_RPM)
#8 RTRIG[5]:R_TRIGs(CLK: L16005_RPM)
#9 R PDO9 <= #10.OUT
#10 RTRIG[16]:R_TRIGs(CLK: #11)
#11 OR(RESET_BOX, MDI_4_0.15)
_END_CFC_
(* the same logic as Structured Text *)
L16001_RPM := ind[1].ALARM;
ind[1](START := L16001_WRK, INPUT := PDI1Q);
RTRIG[1](CLK := L16001_RPM);
IF RTRIG[1].OUT OR RTRIG[2].OUT OR RTRIG[3].OUT OR RTRIG[4].OUT OR RTRIG[5].OUT THEN PDO9 := TRUE; END_IF;
RTRIG[2](CLK := L16106_RPM);
RTRIG[3](CLK := L16201_RPM);
RTRIG[4](CLK := L16101_RPM);
RTRIG[5](CLK := L16005_RPM);
IF RTRIG[16].OUT THEN PDO9 := FALSE; END_IF;
RTRIG[16](CLK := _t46);
_t46 := RESET_BOX OR MDI_4_0.15;
END_PROGRAM

(* POU INIT, ST *)
PROGRAM INIT
VAR
END_VAR
IF eski_counter_1 = 0 THEN
	eski_counter_1 := counter_1;

END_IF;

IF eski_counter_2 = 0 THEN
	eski_counter_2 := counter_2;

END_IF;
IF eski_counter_3 = 0 THEN
	eski_counter_3 := counter_3;

END_IF;

IF eski_counter_4 = 0 THEN
	eski_counter_4 := counter_4;

END_IF;
END_PROGRAM

(* POU mb_read, ST *)
PROGRAM mb_read
VAR
	get1_modbus: MB_RD_HOLD_REGS;    (*функция 03 - чтение параметра типа INT*)
	get2_modbus: MB_RD_INP_REGS;		(*функция 04 - чтение трех параметров типа INT*)
	get3_modbus: MB_RD_HOLD_REGS;	(*функция 03 - чтение параметра типа Float*)

	Buffer: ARRAY[0..255] OF BYTE;		(* байтовый буфер данных *)
     	cmpl: BOOL;
	port_opened:  BYTE := 0;
	Init: BOOL;								(* признак инициализации пользовательской программы *)
	Settings:COMSETTINGS;				(* настройки последовательного порта *)
      	com_num: PORTS:=0;				(*0 - RS-485, 1 - RS-232*)
	enabl: BOOL;							(*состояние работы блока*)
	err: INT;								(*номер ошибки*)
	TimeOut: TIME:=T#50ms;				(*таймаут*)
	Exception: BYTE;
	DataSize: WORD;
	master1: BYTE:= 1;

	t: DWORD;						(*переменная для организации счетчика*)
	A: WORD := 0;					(*счетчик*)
	x:WORD;						(*считанное значение*)
	x1: WORD;						(*переменная для записи по сети*)
	x2: WORD;						(*переменная для записи по сети*)
	x3: WORD;						(*переменная для записи по сети*)
	d:  REAL;						(*считанное значение*)
	ptr_D:POINTER TO BYTE;

	COM_SERVICE1: COM_SERVICE;
END_VAR
(*Организуем счетчик, что бы передавать эти данные по сети*)
t:=t+1;
IF (t MOD 1000)=0 THEN
	A := A + 1;
		IF A > 9999 THEN
			A := 0;
		END_IF
END_IF

(*Устанавливаем настройки COM-порта*)
IF port_opened=0 THEN
		Settings.Port:=com_num;               (*номер COM-порта*)
		Settings.dwBaudRate:=9600;    (*скорость*)
		Settings.byParity:=0;
		Settings.dwTimeout:=0;
		Settings.byStopBits:=0;
		Settings.dwBufferSize:=0;
		Settings.dwScan:=0;
END_IF

COM_SERVICE1(Enable:=(port_opened=0) , Settings:=Settings , Task:=OPEN_TSK  );
(*Если COM-порт открыт, то переходим к приему и передачи данных *)
IF COM_SERVICE1.ready THEN
	port_opened:=2;
END_IF

IF port_opened=2 THEN (*Удачно проинициализировали*)

CASE master1 OF

0: (* функция 03 инт  - ФБ считывает значение параметра  типа int из прибора с адресом 2 в регистр с номером 8 по протоколу Modbus-ASCII*)
get1_modbus(
	Enable:=enabl ,			(* разрешение работы блока *)
	Mode:=MB_ASCII ,		(*режим передачи*)
	DevAddr:=2 ,				(*адрес*)
	FirstAddr:=12 ,				(*номер регистра*)
	Quantity:=1,				(*количество регистров*)
	ComHandle:=Settings.Port , (*номер COM-порта*)
	TimeOut:=TimeOut , 		(*Таймаут T#50ms*)
	Buffer:=Buffer ,			(* буфер данных *)
	Complete=>cmpl ,		(* скопировать признак завершения операции *)
	Exception=>err ,			(* скопировать регистр ошибок *)
	ByteCnt=>DataSize );		(*кол-во считанных байтов *)
(*если установлен признак завершения операции, то *)
IF cmpl THEN
	IF err=0 THEN (*Если нет ошибок, то получаем данные из буфера типа INT*)
		x:=BYTE_TO_WORD(BUFFER[1]) OR SHL(BYTE_TO_WORD(BUFFER[0]),8);
	END_IF
	master1:=1; (*переходим к выполнению следующего ФБ*)
END_IF

1: (* функция 03 флоат - ФБ считывает значение параметра  типа int из прибора с адресом 2 в регистр с номаром 10 по протоколу Modbus-ASCII *)
get3_modbus(
	Enable:=enabl ,			(* разрешение работы блока *)
	Mode:=MB_ASCII ,		(*режим передачи*)
	DevAddr:=2 ,				(*адрес*)
	FirstAddr:=10 ,				(*номер регистра*)
	Quantity:=2,				(*количество регистров*)
	ComHandle:=Settings.Port ,(*номер COM-порта*)
	TimeOut:=TimeOut , 		(*Таймаут T#50ms*)
	Buffer:=Buffer ,			(* буфер данных *)
	Complete=>cmpl ,		(* скопировать признак завершения операции *)
	Exception=>err ,			(* скопировать регистр ошибок *)
	ByteCnt=>DataSize );		(*кол-во считанных байтов *)
(*если установлен признак завершения операции, то *)
IF cmpl THEN
	master1:=2;(*переходим к выполнению следующего ФБ*)
	IF err=0 THEN (*Если нет ошибок, то получаем  данные из буфера типа FLOAT*)
		ptr_D:=ADR(d);
		ptr_D^:=buffer[1];
		ptr_D:=ptr_D+1;
		ptr_D^:=buffer[0];
		ptr_D:=ptr_D+1;
		ptr_D^:=buffer[3];
		ptr_D:=ptr_D+1;
		ptr_D^:=buffer[2];
	END_IF
END_IF

2: (* функция 04 инт - ФБ считывает значения трех параметров типа Int из прибора с адресом 2 начиная с регистра с номeром 12*)
get2_modbus(
	Enable:= enabl,			(* разрешение работы блока *)
	Mode:=MB_ASCII ,		(*режим передачи*)
	DevAddr:=2 ,				(*адрес*)
	FirstAddr:=12 ,				(*номер регистра*)
	Quantity:=6 ,				(*количество регистров*)
	ComHandle:= Settings.Port,(*номер COM-порта*)
	TimeOut:=TimeOut  , 		(*Таймаут T#50ms*)
	Buffer:=Buffer ,			(* буфер данных *)
	Complete=>cmpl ,		(* скопировать признак завершения операции *)
	Exception=>err ,			(* скопировать регистр ошибок *)
	ByteCnt=> DataSize);		(*кол-во считанных байтов *)
(*если установлен признак завершения операции, то *)
IF cmpl THEN
	IF err=0 THEN (*Если нет ошибок, то получаем данные из буфера типа INT*)
		x1:=BYTE_TO_WORD(BUFFER[1]) OR SHL(BYTE_TO_WORD(BUFFER[0]),8);
		x2:=BYTE_TO_WORD(BUFFER[5]) OR SHL(BYTE_TO_WORD(BUFFER[4]),8);
		x3:=BYTE_TO_WORD(BUFFER[9]) OR SHL(BYTE_TO_WORD(BUFFER[8]),8);
	END_IF
	master1:=0;(*переходим к выполнению следующего ФБ*)
END_IF
END_CASE

IF  enabl = FALSE THEN
 	enabl := TRUE;
END_IF

IF  err <> 0 THEN
 	enabl := FALSE;
END_IF

END_IF
END_PROGRAM

(* POU mb_write, ST *)
PROGRAM mb_write
VAR
	send1_modbus:MB_WR_SNG_REG; (*функция 06 - запись параметра*)
	send2_modbus: MB_WR_REGS;         (*функция 16 - запись параметров*)
	COM_SERVICE1: COM_SERVICE;	   (*ФБ открытия порта*)

	Buffer: ARRAY[0..255] OF BYTE;		(* байтовый буфер данных *)
     	cmpl: BOOL;							(* признак завершения операции *)
	port_opened:  BYTE := 0;				(*состояние порта*)
	Init: BOOL;								(* признак инициализации пользовательской программы *)
	Settings:COMSETTINGS;				(* настройки последовательного порта *)
      	com_num: PORTS:=0;				(*0 - RS-485, 1 - RS-232*)
	enabl: BOOL;							(*состояние работы блока*)
	err: INT;								(*номер ошибки*)
	TimeOut: TIME:=T#50ms;				(*таймаут*)
	Exception: BYTE;
	DataSize: WORD;
	master1: BYTE;

	t: DWORD;					(*переменная для организации счетчика*)
	A: WORD := 0;				(*счетчик*)
	f1:DINT:=65;				(*Записываемый параметр типа DINT*)
	f2:REAL:=12.7;			(*Записываемый параметр типа REAL*)
	ptr_f2:POINTER TO BYTE;

END_VAR
(*Организуем счетчик, что бы передавать эти данные по сети*)
t:=t+1;
IF (t MOD 1000)=0 THEN
	A := A + 1;
		IF A > 9999 THEN
			A := 0;
		END_IF
END_IF

(*Устанавливаем настройки COM-порта*)
IF port_opened=0 THEN
		Settings.Port:=com_num;               (*номер COM-порта*)
		Settings.dwBaudRate:=9600;    (*скорость*)
		Settings.byParity:=0;
		Settings.dwTimeout:=0;
		Settings.byStopBits:=0;
		Settings.dwBufferSize:=0;
		Settings.dwScan:=0;
END_IF

(*Открываем COM-порт*)
COM_SERVICE1(Enable:=(port_opened=0) , Settings:=Settings , Task:=OPEN_TSK  );
(*Если COM-порт открыт, то переходим к приему и передачи данных *)
IF COM_SERVICE1.ready THEN
	port_opened:=2;
END_IF

IF port_opened=2 THEN (*Удачно проинициализировали*)

CASE master1 OF

0:  (* функция 06  - запись параметра типа Int в прибор с адресом 1 в регистр 0*)
send1_modbus(
	Enable:=enabl ,				(* разрешение работы блока *)
	Mode:=MB_RTU ,			(*режим передачи*)
	DevAddr:=2 ,					(*адрес*)
	RegAddr:=6 ,					(*регистр*)
	Value:=A,						(*значение переменной, которое надо передать*)
      ComHandle:= Settings.Port, 	(*номер сом-порта*)
	TimeOut:=TimeOut ,			(*таймаут T#50ms*)
	Complete=>cmpl ,			(* скопировать признак завершения операции *)
	Exception=>err );				(* скопировать регистр ошибок *)
(*если установлен признак завершения операции, то *)
IF cmpl THEN
	master1:=1; (*переходим к выполнению следующего блока*)
END_IF

1: (* функция 16  - запись параметров типа Int (регистр 4) и Real (регистр 6) в прибор с адресом 2 *)
(*запись в буффер параметра типа INT*)
Buffer[1] := DINT_TO_BYTE(f1);
Buffer[0] := DINT_TO_BYTE( SHR(f1,8));
Buffer[3] := DINT_TO_BYTE( SHR(f1,16));
Buffer[2] := DINT_TO_BYTE( SHR(f1,24));

(*запись в буффер параметра типа Float*)
ptr_f2:=ADR(f2);
     buffer[5] := ptr_f2^;
     ptr_f2:=ptr_f2+1;
     buffer[4] := ptr_f2^;
     ptr_f2:=ptr_f2+1;
     buffer[7] := ptr_f2^;
     ptr_f2:=ptr_f2+1;
     buffer[6] := ptr_f2^;

send2_modbus(
	Enable:= enabl,			(* разрешение работы блока *)
	Mode:=MB_RTU ,		(*режим передачи*)
	DevAddr:=2 , 				(*адрес*)
	FirstAddr:= 4, 				(*номер регистра*)
	Quantity:= 4,   				(*количество записываемых регистров*)
	ComHandle:=Settings.Port ,(*номер сом-порта*)
	TimeOut:=TimeOut ,		(*таймаут T#50ms*)
	Buffer:=Buffer ,			(* буфер данных *)
	Complete=>cmpl ,		(* скопировать признак завершения операции *)
	Exception=>err ,			(* скопировать регистр ошибок *)
	RegCnt=> DataSize);		(*кол-во считанных байтов *)
(*если установлен признак завершения операции, то *)
IF cmpl THEN
	master1:=0;(*переходим к выполнению следующего блока*)
END_IF

END_CASE

IF  enabl = FALSE THEN
 	enabl := TRUE;
END_IF
IF  err <> 0 THEN
 	enabl := FALSE;
END_IF

END_IF
END_PROGRAM

(* POU SUCTION_CMD, SFC *)
FUNCTION_BLOCK SUCTION_CMD
VAR_INPUT
	EN : BOOL;

END_VAR
VAR_IN_OUT
	STOP : BOOL;
	START : BOOL;
END_VAR

VAR
	T : BOOL;
END_VAR
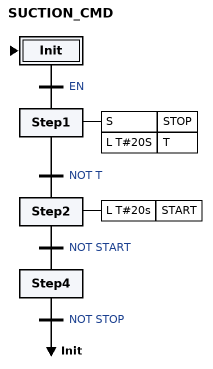
INITIAL_STEP Init:
END_STEP
TRANSITION FROM Init TO Step1 := EN;
END_TRANSITION
STEP Step1:
	STOP(S);
	T(L, T#20S);
END_STEP
TRANSITION FROM Step1 TO Step2 := NOT T;
END_TRANSITION
STEP Step2:
	START(L, T#20s);
END_STEP
TRANSITION FROM Step2 TO Step4 := NOT START;
END_TRANSITION
STEP Step4:
END_STEP
TRANSITION FROM Step4 TO Init := NOT STOP;
END_TRANSITION
END_FUNCTION_BLOCK
